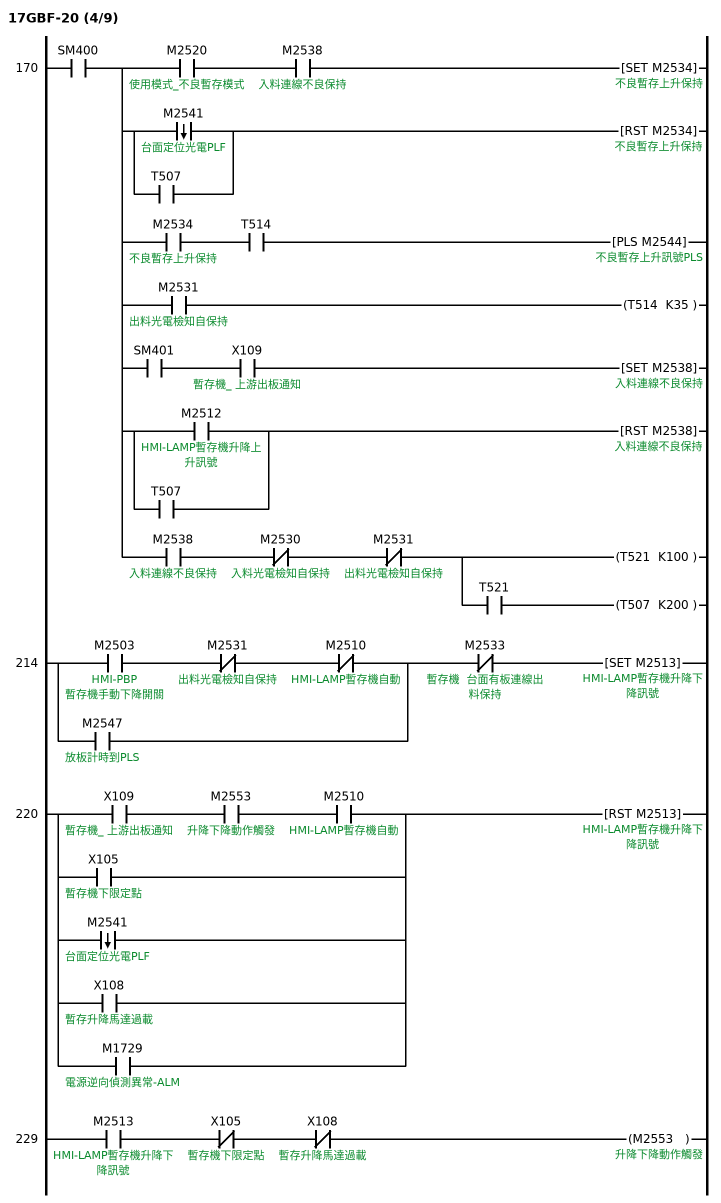
[picture p144: ladder of 17GBF-20, rungs at steps 170 to 229]
170   LD      SM400
      MPS
      AND     M2520  ; 使用模式_不良暫存模式
      AND     M2538  ; 入料連線不良保持
      SET     M2534  ; 不良暫存上升保持
      MRD
      LDF     M2541  ; 台面定位光電PLF
      OR      T507
      ANB
      RST     M2534  ; 不良暫存上升保持
      MRD
      AND     M2534  ; 不良暫存上升保持
      AND     T514
      PLS     M2544  ; 不良暫存上升訊號PLS
      MRD
      AND     M2531  ; 出料光電檢知自保持
      OUT     T514 K35
      MRD
      AND     SM401
      AND     X109  ; 暫存機_ 上游出板通知
      SET     M2538  ; 入料連線不良保持
      MRD
      LD      M2512  ; HMI-LAMP暫存機升降上升訊號
      OR      T507
      ANB
      RST     M2538  ; 入料連線不良保持
      MPP
      AND     M2538  ; 入料連線不良保持
      ANI     M2530  ; 入料光電檢知自保持
      ANI     M2531  ; 出料光電檢知自保持
      OUT     T521 K100
      AND     T521
      OUT     T507 K200
214   LD      M2503  ; HMI-PBP 暫存機手動下降開關
      ANI     M2531  ; 出料光電檢知自保持
      ANI     M2510  ; HMI-LAMP暫存機自動
      OR      M2547  ; 放板計時到PLS
      ANI     M2533  ; 暫存機  台面有板連線出料保持
      SET     M2513  ; HMI-LAMP暫存機升降下降訊號
220   LD      X109  ; 暫存機_ 上游出板通知
      AND     M2553  ; 升降下降動作觸發
      AND     M2510  ; HMI-LAMP暫存機自動
      OR      X105  ; 暫存機下限定點
      ORF     M2541  ; 台面定位光電PLF
      OR      X108  ; 暫存升降馬達過載
      OR      M1729  ; 電源逆向偵測異常-ALM
      RST     M2513  ; HMI-LAMP暫存機升降下降訊號
229   LD      M2513  ; HMI-LAMP暫存機升降下降訊號
      ANI     X105  ; 暫存機下限定點
      ANI     X108  ; 暫存升降馬達過載
      OUT     M2553  ; 升降下降動作觸發
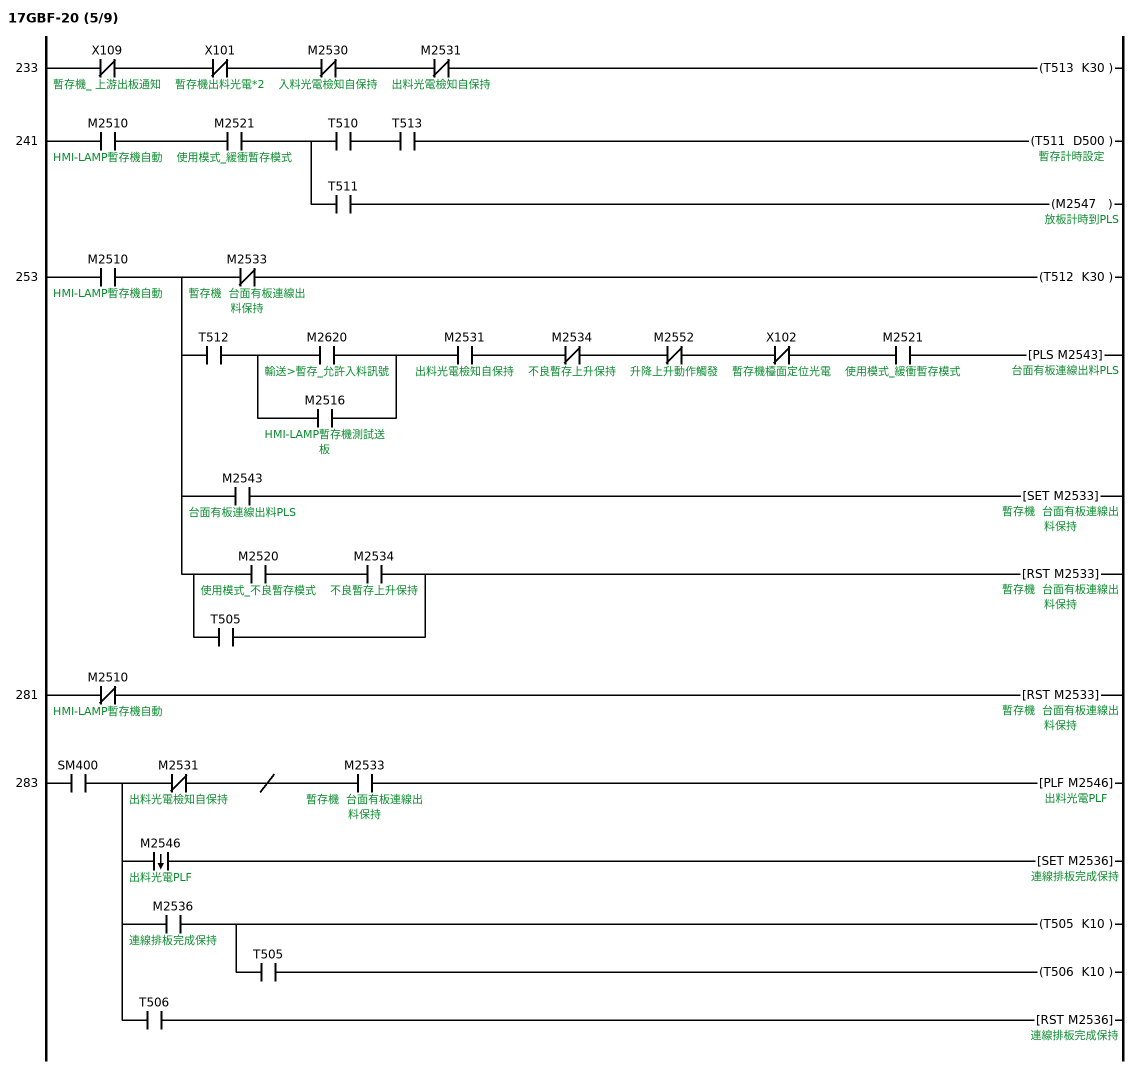
233   LDI     X109  ; 暫存機_ 上游出板通知
      ANI     X101  ; 暫存機出料光電*2
      ANI     M2530  ; 入料光電檢知自保持
      ANI     M2531  ; 出料光電檢知自保持
      OUT     T513 K30
241   LD      M2510  ; HMI-LAMP暫存機自動
      AND     M2521  ; 使用模式_緩衝暫存模式
      MPS
      AND     T510
      AND     T513
      OUT     T511 D500  ; 暫存計時設定
      MPP
      AND     T511
      OUT     M2547  ; 放板計時到PLS
253   LD      M2510  ; HMI-LAMP暫存機自動
      MPS
      ANI     M2533  ; 暫存機  台面有板連線出料保持
      OUT     T512 K30
      MRD
      AND     T512
      LD      M2620  ; 輸送>暫存_允許入料訊號
      OR      M2516  ; HMI-LAMP暫存機測試送板
      ANB
      AND     M2531  ; 出料光電檢知自保持
      ANI     M2534  ; 不良暫存上升保持
      ANI     M2552  ; 升降上升動作觸發
      ANI     X102  ; 暫存機檯面定位光電
      AND     M2521  ; 使用模式_緩衝暫存模式
      PLS     M2543  ; 台面有板連線出料PLS
      MRD
      AND     M2543  ; 台面有板連線出料PLS
      SET     M2533  ; 暫存機  台面有板連線出料保持
      MPP
      LD      M2520  ; 使用模式_不良暫存模式
      AND     M2534  ; 不良暫存上升保持
      OR      T505
      ANB
      RST     M2533  ; 暫存機  台面有板連線出料保持
281   LDI     M2510  ; HMI-LAMP暫存機自動
      RST     M2533  ; 暫存機  台面有板連線出料保持
283   LD      SM400
      MPS
      ANI     M2531  ; 出料光電檢知自保持
      INV
      AND     M2533  ; 暫存機  台面有板連線出料保持
      PLF     M2546  ; 出料光電PLF
      MRD
      ANDF    M2546  ; 出料光電PLF
      SET     M2536  ; 連線排板完成保持
      MRD
      AND     M2536  ; 連線排板完成保持
      OUT     T505 K10
      AND     T505
      OUT     T506 K10
      MPP
      AND     T506
      RST     M2536  ; 連線排板完成保持
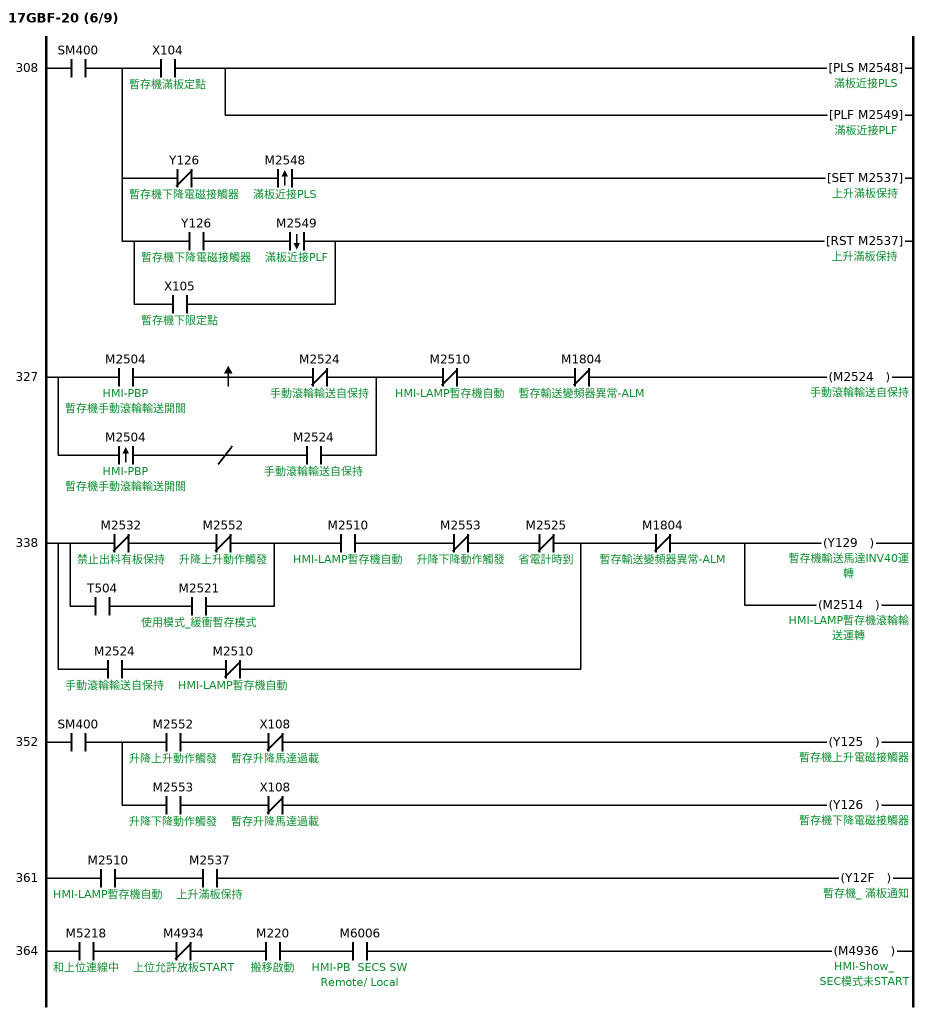
308   LD      SM400
      MPS
      AND     X104  ; 暫存機滿板定點
      PLS     M2548  ; 滿板近接PLS
      PLF     M2549  ; 滿板近接PLF
      MRD
      ANI     Y126  ; 暫存機下降電磁接觸器
      ANDP    M2548  ; 滿板近接PLS
      SET     M2537  ; 上升滿板保持
      MPP
      LD      Y126  ; 暫存機下降電磁接觸器
      ANDF    M2549  ; 滿板近接PLF
      OR      X105  ; 暫存機下限定點
      ANB
      RST     M2537  ; 上升滿板保持
327   LD      M2504  ; HMI-PBP 暫存機手動滾輪輸送開關
      MEP
      ANI     M2524  ; 手動滾輪輸送自保持
      LDP     M2504  ; HMI-PBP 暫存機手動滾輪輸送開關
      INV
      AND     M2524  ; 手動滾輪輸送自保持
      ORB
      ANI     M2510  ; HMI-LAMP暫存機自動
      ANI     M1804  ; 暫存輸送變頻器異常-ALM
      OUT     M2524  ; 手動滾輪輸送自保持
338   LDI     M2532  ; 禁止出料有板保持
      ANI     M2552  ; 升降上升動作觸發
      LD      T504
      AND     M2521  ; 使用模式_緩衝暫存模式
      ORB
      AND     M2510  ; HMI-LAMP暫存機自動
      ANI     M2553  ; 升降下降動作觸發
      ANI     M2525  ; 省電計時到
      LD      M2524  ; 手動滾輪輸送自保持
      ANI     M2510  ; HMI-LAMP暫存機自動
      ORB
      ANI     M1804  ; 暫存輸送變頻器異常-ALM
      OUT     Y129  ; 暫存機輸送馬達INV40運轉
      OUT     M2514  ; HMI-LAMP暫存機滾輪輸送運轉
352   LD      SM400
      MPS
      AND     M2552  ; 升降上升動作觸發
      ANI     X108  ; 暫存升降馬達過載
      OUT     Y125  ; 暫存機上升電磁接觸器
      MPP
      AND     M2553  ; 升降下降動作觸發
      ANI     X108  ; 暫存升降馬達過載
      OUT     Y126  ; 暫存機下降電磁接觸器
361   LD      M2510  ; HMI-LAMP暫存機自動
      AND     M2537  ; 上升滿板保持
      OUT     Y12F  ; 暫存機_ 滿板通知
364   LD      M5218  ; 和上位連線中
      ANI     M4934  ; 上位允許放板START
      AND     M220  ; 搬移啟動
      AND     M6006  ; HMI-PB  SECS SW  Remote/ Local
      OUT     M4936  ; HMI-Show_SEC模式未START
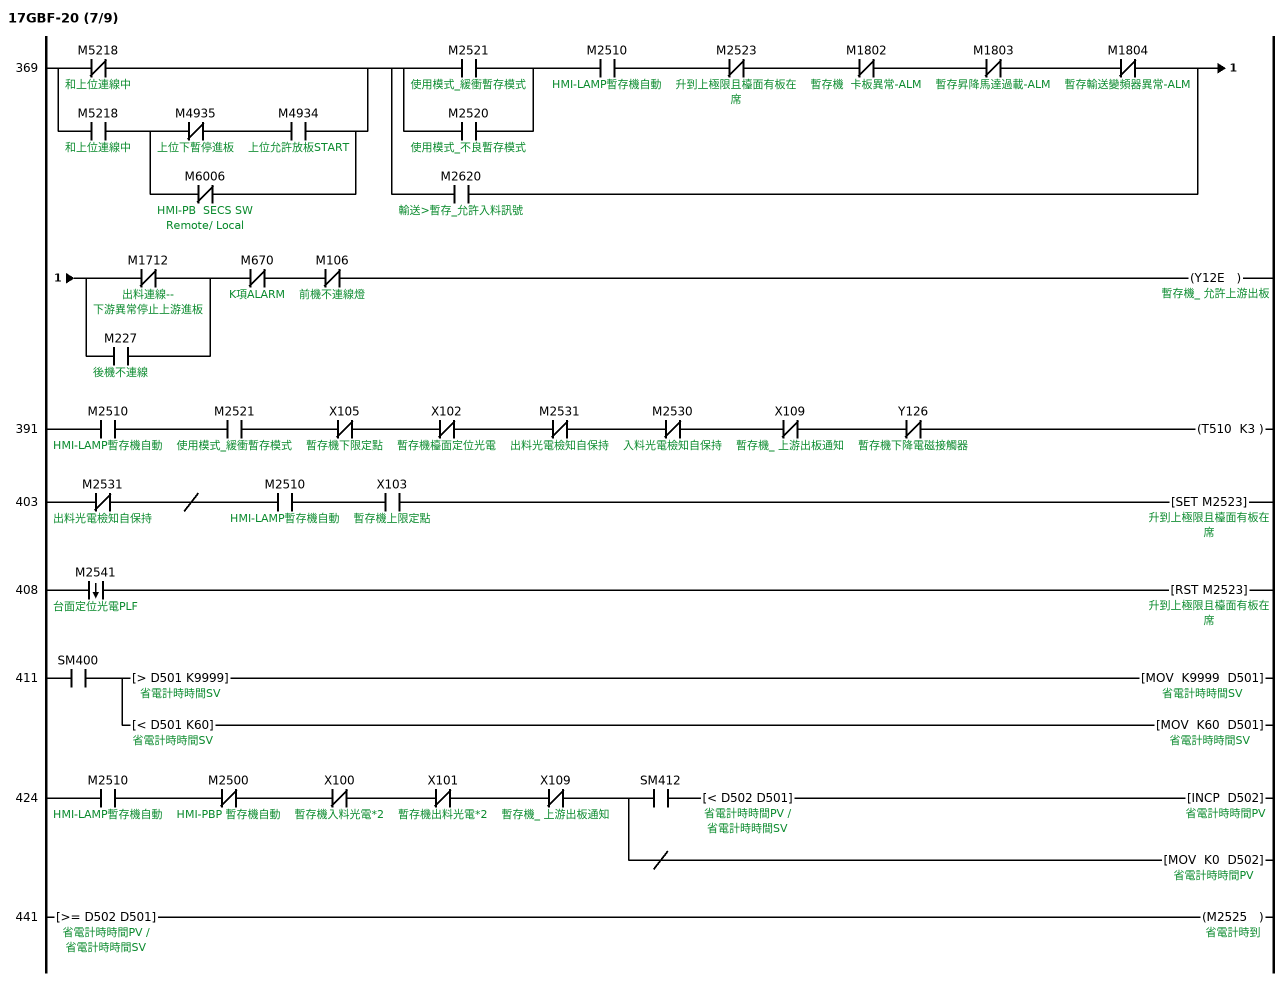
369   LDI     M5218  ; 和上位連線中
      LD      M5218  ; 和上位連線中
      LDI     M4935  ; 上位下暫停進板
      AND     M4934  ; 上位允許放板START
      ORI     M6006  ; HMI-PB  SECS SW  Remote/ Local
      ANB
      ORB
      LD      M2521  ; 使用模式_緩衝暫存模式
      OR      M2520  ; 使用模式_不良暫存模式
      AND     M2510  ; HMI-LAMP暫存機自動
      ANI     M2523  ; 升到上極限且檯面有板在席
      ANI     M1802  ; 暫存機  卡板異常-ALM
      ANI     M1803  ; 暫存昇降馬達過載-ALM
      ANI     M1804  ; 暫存輸送變頻器異常-ALM
      OR      M2620  ; 輸送>暫存_允許入料訊號
      ANB
      LDI     M1712  ; 出料連線--下游異常停止上游進板
      OR      M227  ; 後機不連線
      ANB
      ANI     M670  ; K項ALARM
      ANI     M106  ; 前機不連線燈
      OUT     Y12E  ; 暫存機_ 允許上游出板
391   LD      M2510  ; HMI-LAMP暫存機自動
      AND     M2521  ; 使用模式_緩衝暫存模式
      ANI     X105  ; 暫存機下限定點
      ANI     X102  ; 暫存機檯面定位光電
      ANI     M2531  ; 出料光電檢知自保持
      ANI     M2530  ; 入料光電檢知自保持
      ANI     X109  ; 暫存機_ 上游出板通知
      ANI     Y126  ; 暫存機下降電磁接觸器
      OUT     T510 K3
403   LDI     M2531  ; 出料光電檢知自保持
      INV
      AND     M2510  ; HMI-LAMP暫存機自動
      AND     X103  ; 暫存機上限定點
      SET     M2523  ; 升到上極限且檯面有板在席
408   LDF     M2541  ; 台面定位光電PLF
      RST     M2523  ; 升到上極限且檯面有板在席
411   LD      SM400
      MPS
      AND>    D501 K9999  ; 省電計時時間SV
      MOV     K9999 D501
      MPP
      AND<    D501 K60  ; 省電計時時間SV
      MOV     K60 D501
424   LD      M2510  ; HMI-LAMP暫存機自動
      ANI     M2500  ; HMI-PBP 暫存機自動
      ANI     X100  ; 暫存機入料光電*2
      ANI     X101  ; 暫存機出料光電*2
      ANI     X109  ; 暫存機_ 上游出板通知
      MPS
      AND     SM412
      AND<    D502 D501  ; 省電計時時間PV / 省電計時時間SV
      INCP    D502
      MPP
      INV
      MOV     K0 D502
441   LD>=    D502 D501  ; 省電計時時間PV / 省電計時時間SV
      OUT     M2525  ; 省電計時到
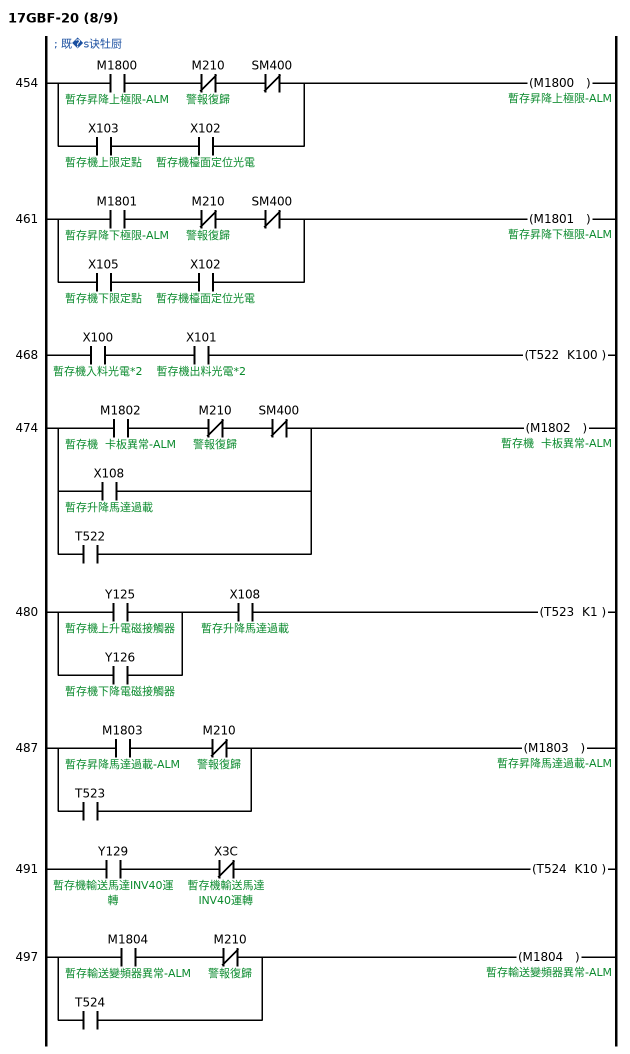
; 暫存機警報
454   LD      M1800  ; 暫存昇降上極限-ALM
      ANI     M210  ; 警報復歸
      ANI     SM400
      LD      X103  ; 暫存機上限定點
      AND     X102  ; 暫存機檯面定位光電
      ORB
      OUT     M1800  ; 暫存昇降上極限-ALM
461   LD      M1801  ; 暫存昇降下極限-ALM
      ANI     M210  ; 警報復歸
      ANI     SM400
      LD      X105  ; 暫存機下限定點
      AND     X102  ; 暫存機檯面定位光電
      ORB
      OUT     M1801  ; 暫存昇降下極限-ALM
468   LD      X100  ; 暫存機入料光電*2
      AND     X101  ; 暫存機出料光電*2
      OUT     T522 K100
474   LD      M1802  ; 暫存機  卡板異常-ALM
      ANI     M210  ; 警報復歸
      ANI     SM400
      OR      X108  ; 暫存升降馬達過載
      OR      T522
      OUT     M1802  ; 暫存機  卡板異常-ALM
480   LD      Y125  ; 暫存機上升電磁接觸器
      OR      Y126  ; 暫存機下降電磁接觸器
      AND     X108  ; 暫存升降馬達過載
      OUT     T523 K1
487   LD      M1803  ; 暫存昇降馬達過載-ALM
      ANI     M210  ; 警報復歸
      OR      T523
      OUT     M1803  ; 暫存昇降馬達過載-ALM
491   LD      Y129  ; 暫存機輸送馬達INV40運轉
      ANI     X3C  ; 暫存機輸送馬達  INV40運轉
      OUT     T524 K10
497   LD      M1804  ; 暫存輸送變頻器異常-ALM
      ANI     M210  ; 警報復歸
      OR      T524
      OUT     M1804  ; 暫存輸送變頻器異常-ALM
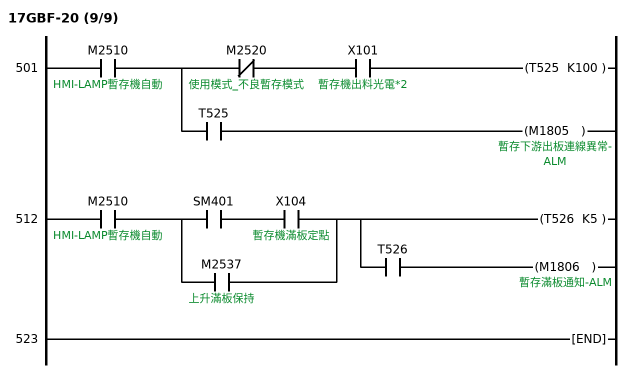
501   LD      M2510  ; HMI-LAMP暫存機自動
      MPS
      ANI     M2520  ; 使用模式_不良暫存模式
      AND     X101  ; 暫存機出料光電*2
      OUT     T525 K100
      MPP
      AND     T525
      OUT     M1805  ; 暫存下游出板連線異常-ALM
512   LD      M2510  ; HMI-LAMP暫存機自動
      LD      SM401
      AND     X104  ; 暫存機滿板定點
      OR      M2537  ; 上升滿板保持
      ANB
      OUT     T526 K5
      AND     T526
      OUT     M1806  ; 暫存滿板通知-ALM
523   END
END_PROGRAM

PROGRAM 18GCV
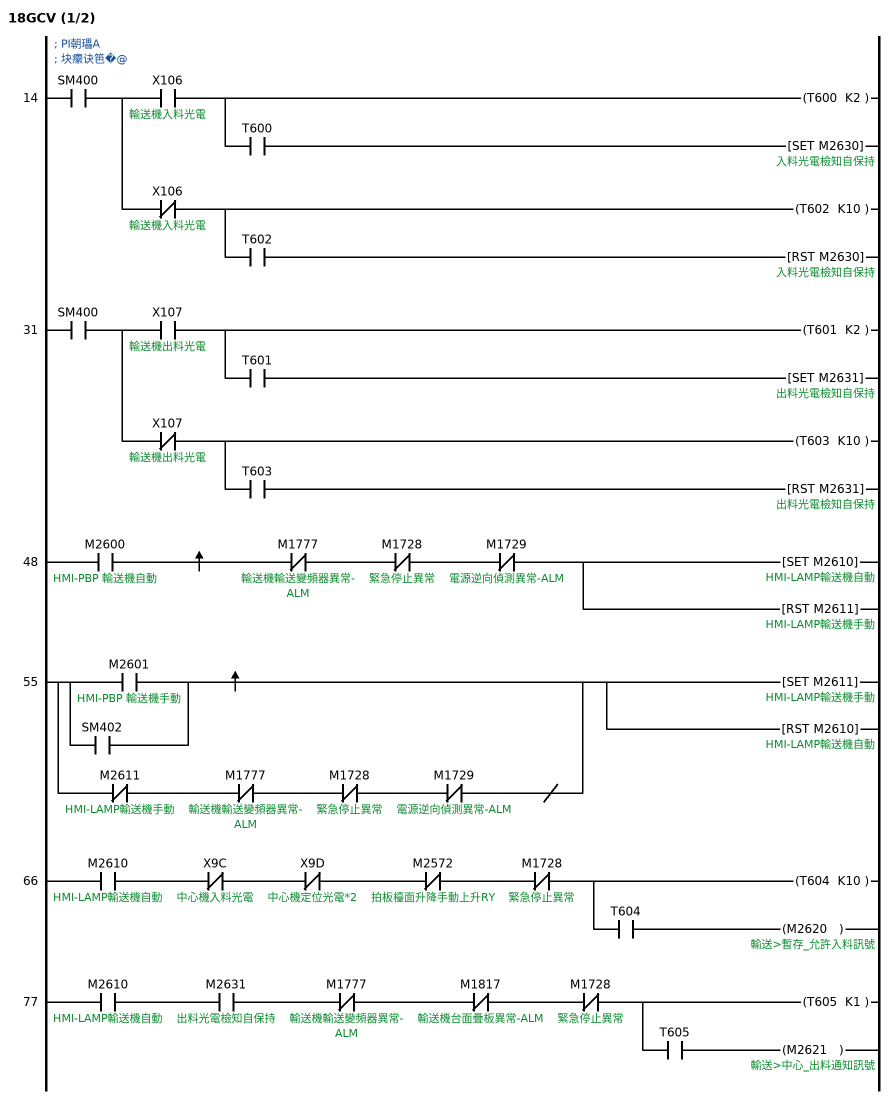
; PI朝瓃Α
; 輸送機動作
14    LD      SM400
      MPS
      AND     X106  ; 輸送機入料光電
      OUT     T600 K2
      AND     T600
      SET     M2630  ; 入料光電檢知自保持
      MPP
      ANI     X106  ; 輸送機入料光電
      OUT     T602 K10
      AND     T602
      RST     M2630  ; 入料光電檢知自保持
31    LD      SM400
      MPS
      AND     X107  ; 輸送機出料光電
      OUT     T601 K2
      AND     T601
      SET     M2631  ; 出料光電檢知自保持
      MPP
      ANI     X107  ; 輸送機出料光電
      OUT     T603 K10
      AND     T603
      RST     M2631  ; 出料光電檢知自保持
48    LD      M2600  ; HMI-PBP 輸送機自動
      MEP
      ANI     M1777  ; 輸送機輸送變頻器異常-ALM
      ANI     M1728  ; 緊急停止異常
      ANI     M1729  ; 電源逆向偵測異常-ALM
      SET     M2610  ; HMI-LAMP輸送機自動
      RST     M2611  ; HMI-LAMP輸送機手動
55    LD      M2601  ; HMI-PBP 輸送機手動
      OR      SM402
      MEP
      LDI     M2611  ; HMI-LAMP輸送機手動
      ANI     M1777  ; 輸送機輸送變頻器異常-ALM
      ANI     M1728  ; 緊急停止異常
      ANI     M1729  ; 電源逆向偵測異常-ALM
      INV
      ORB
      SET     M2611  ; HMI-LAMP輸送機手動
      RST     M2610  ; HMI-LAMP輸送機自動
66    LD      M2610  ; HMI-LAMP輸送機自動
      ANI     X9C  ; 中心機入料光電
      ANI     X9D  ; 中心機定位光電*2
      ANI     M2572  ; 拍板檯面升降手動上升RY
      ANI     M1728  ; 緊急停止異常
      OUT     T604 K10
      AND     T604
      OUT     M2620  ; 輸送>暫存_允許入料訊號
77    LD      M2610  ; HMI-LAMP輸送機自動
      AND     M2631  ; 出料光電檢知自保持
      ANI     M1777  ; 輸送機輸送變頻器異常-ALM
      ANI     M1817  ; 輸送機台面疊板異常-ALM
      ANI     M1728  ; 緊急停止異常
      OUT     T605 K1
      AND     T605
      OUT     M2621  ; 輸送>中心_出料通知訊號
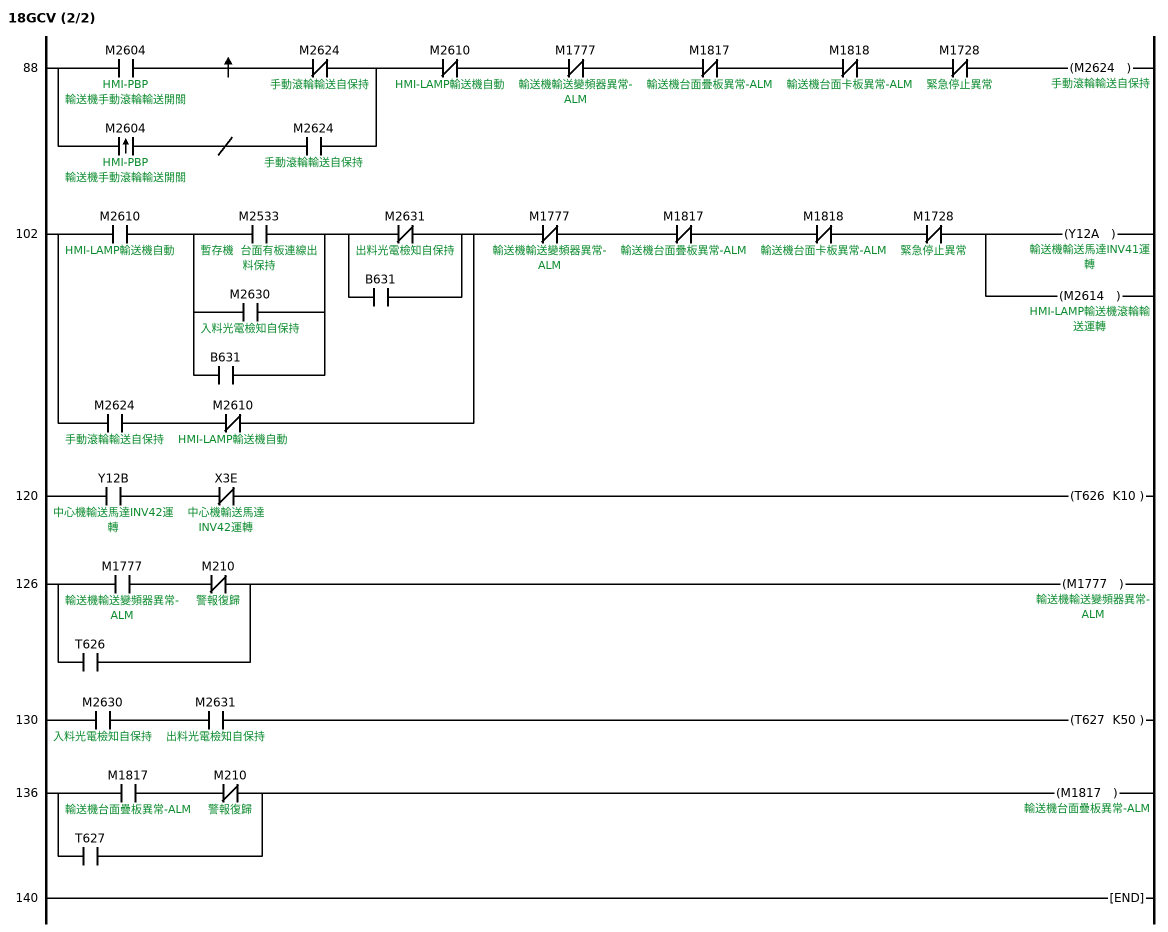
88    LD      M2604  ; HMI-PBP 輸送機手動滾輪輸送開關
      MEP
      ANI     M2624  ; 手動滾輪輸送自保持
      LDP     M2604  ; HMI-PBP 輸送機手動滾輪輸送開關
      INV
      AND     M2624  ; 手動滾輪輸送自保持
      ORB
      ANI     M2610  ; HMI-LAMP輸送機自動
      ANI     M1777  ; 輸送機輸送變頻器異常-ALM
      ANI     M1817  ; 輸送機台面疊板異常-ALM
      ANI     M1818  ; 輸送機台面卡板異常-ALM
      ANI     M1728  ; 緊急停止異常
      OUT     M2624  ; 手動滾輪輸送自保持
102   LD      M2610  ; HMI-LAMP輸送機自動
      LD      M2533  ; 暫存機  台面有板連線出料保持
      OR      M2630  ; 入料光電檢知自保持
      OR      B631
      ANB
      LDI     M2631  ; 出料光電檢知自保持
      OR      B631
      ANB
      LD      M2624  ; 手動滾輪輸送自保持
      ANI     M2610  ; HMI-LAMP輸送機自動
      ORB
      ANI     M1777  ; 輸送機輸送變頻器異常-ALM
      ANI     M1817  ; 輸送機台面疊板異常-ALM
      ANI     M1818  ; 輸送機台面卡板異常-ALM
      ANI     M1728  ; 緊急停止異常
      OUT     Y12A  ; 輸送機輸送馬達INV41運轉
      OUT     M2614  ; HMI-LAMP輸送機滾輪輸送運轉
120   LD      Y12B  ; 中心機輸送馬達INV42運轉
      ANI     X3E  ; 中心機輸送馬達  INV42運轉
      OUT     T626 K10
126   LD      M1777  ; 輸送機輸送變頻器異常-ALM
      ANI     M210  ; 警報復歸
      OR      T626
      OUT     M1777  ; 輸送機輸送變頻器異常-ALM
130   LD      M2630  ; 入料光電檢知自保持
      AND     M2631  ; 出料光電檢知自保持
      OUT     T627 K50
136   LD      M1817  ; 輸送機台面疊板異常-ALM
      ANI     M210  ; 警報復歸
      OR      T627
      OUT     M1817  ; 輸送機台面疊板異常-ALM
140   END
END_PROGRAM

PROGRAM 19GTC-7
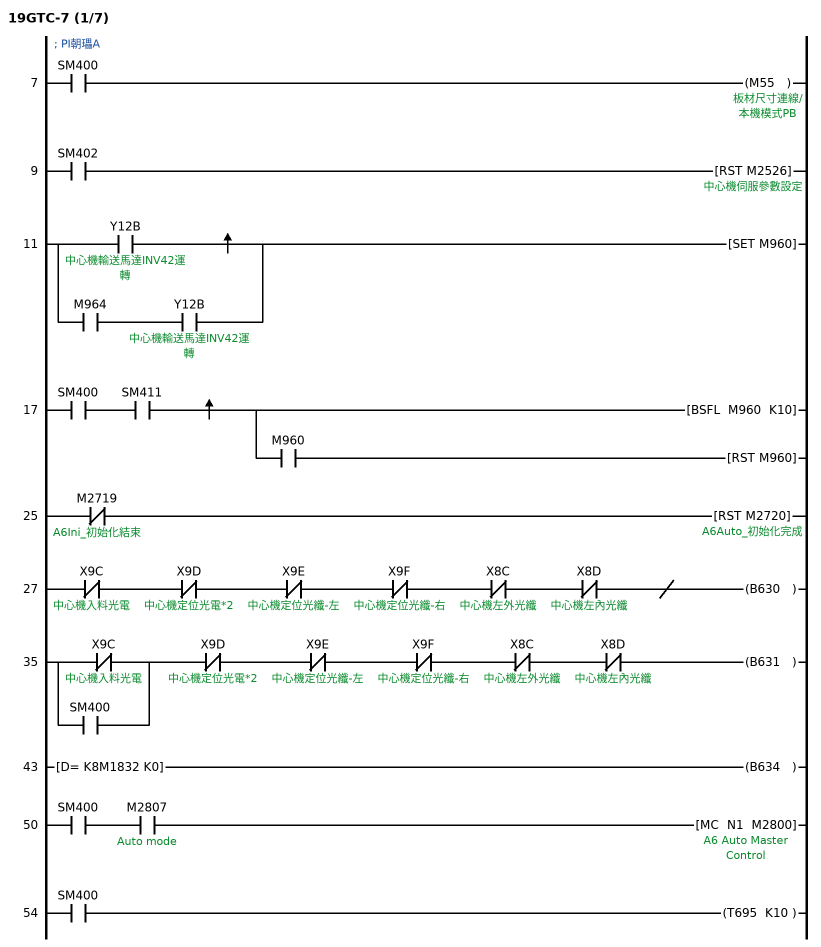
; PI朝瓃Α
7     LD      SM400
      OUT     M55  ; 板材尺寸連線/本機模式PB
9     LD      SM402
      RST     M2526  ; 中心機伺服參數設定
11    LD      Y12B  ; 中心機輸送馬達INV42運轉
      MEP
      LD      M964
      AND     Y12B  ; 中心機輸送馬達INV42運轉
      ORB
      SET     M960
17    LD      SM400
      AND     SM411
      MEP
      BSFL    M960 K10
      AND     M960
      RST     M960
25    LDI     M2719  ; A6Ini_初始化結束
      RST     M2720  ; A6Auto_初始化完成
27    LDI     X9C  ; 中心機入料光電
      ANI     X9D  ; 中心機定位光電*2
      ANI     X9E  ; 中心機定位光纖-左
      ANI     X9F  ; 中心機定位光纖-右
      ANI     X8C  ; 中心機左外光纖
      ANI     X8D  ; 中心機左內光纖
      INV
      OUT     B630
35    LDI     X9C  ; 中心機入料光電
      OR      SM400
      ANI     X9D  ; 中心機定位光電*2
      ANI     X9E  ; 中心機定位光纖-左
      ANI     X9F  ; 中心機定位光纖-右
      ANI     X8C  ; 中心機左外光纖
      ANI     X8D  ; 中心機左內光纖
      OUT     B631
43    LDD=    K8M1832 K0
      OUT     B634
50    LD      SM400
      AND     M2807  ; Auto mode
      MC      N1 M2800  ; A6 Auto Master Control
54    LD      SM400
      OUT     T695 K10
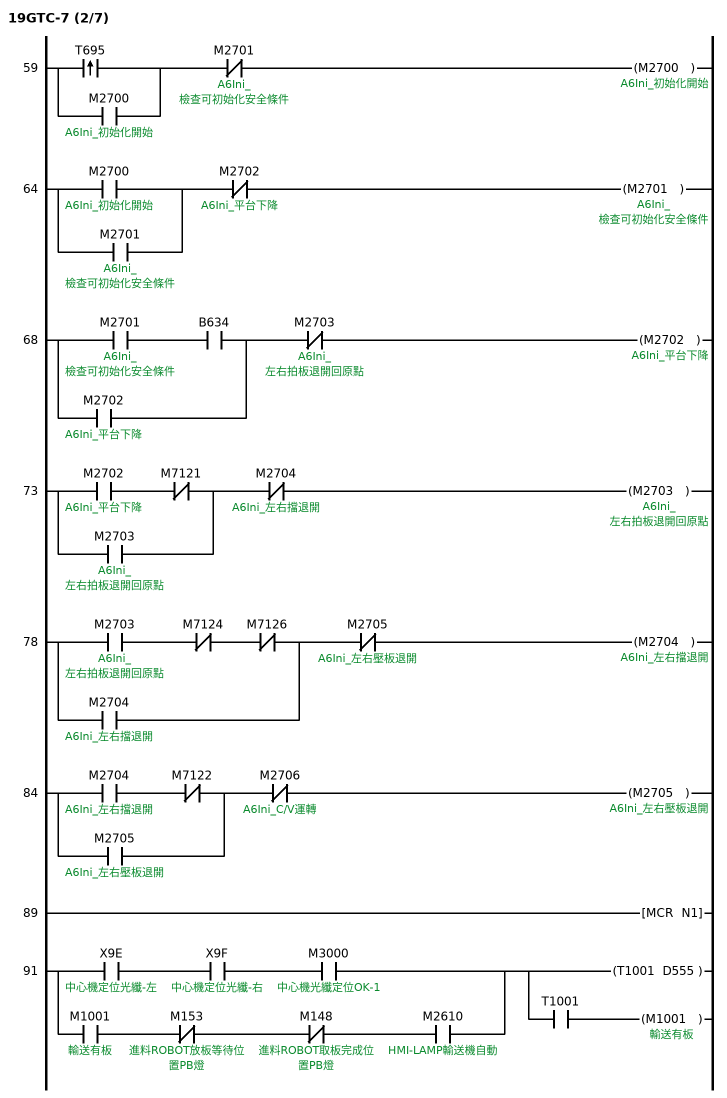
59    LDP     T695
      OR      M2700  ; A6Ini_初始化開始
      ANI     M2701  ; A6Ini_檢查可初始化安全條件
      OUT     M2700  ; A6Ini_初始化開始
64    LD      M2700  ; A6Ini_初始化開始
      OR      M2701  ; A6Ini_檢查可初始化安全條件
      ANI     M2702  ; A6Ini_平台下降
      OUT     M2701  ; A6Ini_檢查可初始化安全條件
68    LD      M2701  ; A6Ini_檢查可初始化安全條件
      AND     B634
      OR      M2702  ; A6Ini_平台下降
      ANI     M2703  ; A6Ini_左右拍板退開回原點
      OUT     M2702  ; A6Ini_平台下降
73    LD      M2702  ; A6Ini_平台下降
      ANI     M7121
      OR      M2703  ; A6Ini_左右拍板退開回原點
      ANI     M2704  ; A6Ini_左右擋退開
      OUT     M2703  ; A6Ini_左右拍板退開回原點
78    LD      M2703  ; A6Ini_左右拍板退開回原點
      ANI     M7124
      ANI     M7126
      OR      M2704  ; A6Ini_左右擋退開
      ANI     M2705  ; A6Ini_左右壓板退開
      OUT     M2704  ; A6Ini_左右擋退開
84    LD      M2704  ; A6Ini_左右擋退開
      ANI     M7122
      OR      M2705  ; A6Ini_左右壓板退開
      ANI     M2706  ; A6Ini_C/V運轉
      OUT     M2705  ; A6Ini_左右壓板退開
89    MCR     N1
91    LD      X9E  ; 中心機定位光纖-左
      AND     X9F  ; 中心機定位光纖-右
      AND     M3000  ; 中心機光纖定位OK-1
      LD      M1001  ; 輸送有板
      ANI     M153  ; 進料ROBOT放板等待位置PB燈
      ANI     M148  ; 進料ROBOT取板完成位置PB燈
      AND     M2610  ; HMI-LAMP輸送機自動
      ORB
      OUT     T1001 D555
      AND     T1001
      OUT     M1001  ; 輸送有板
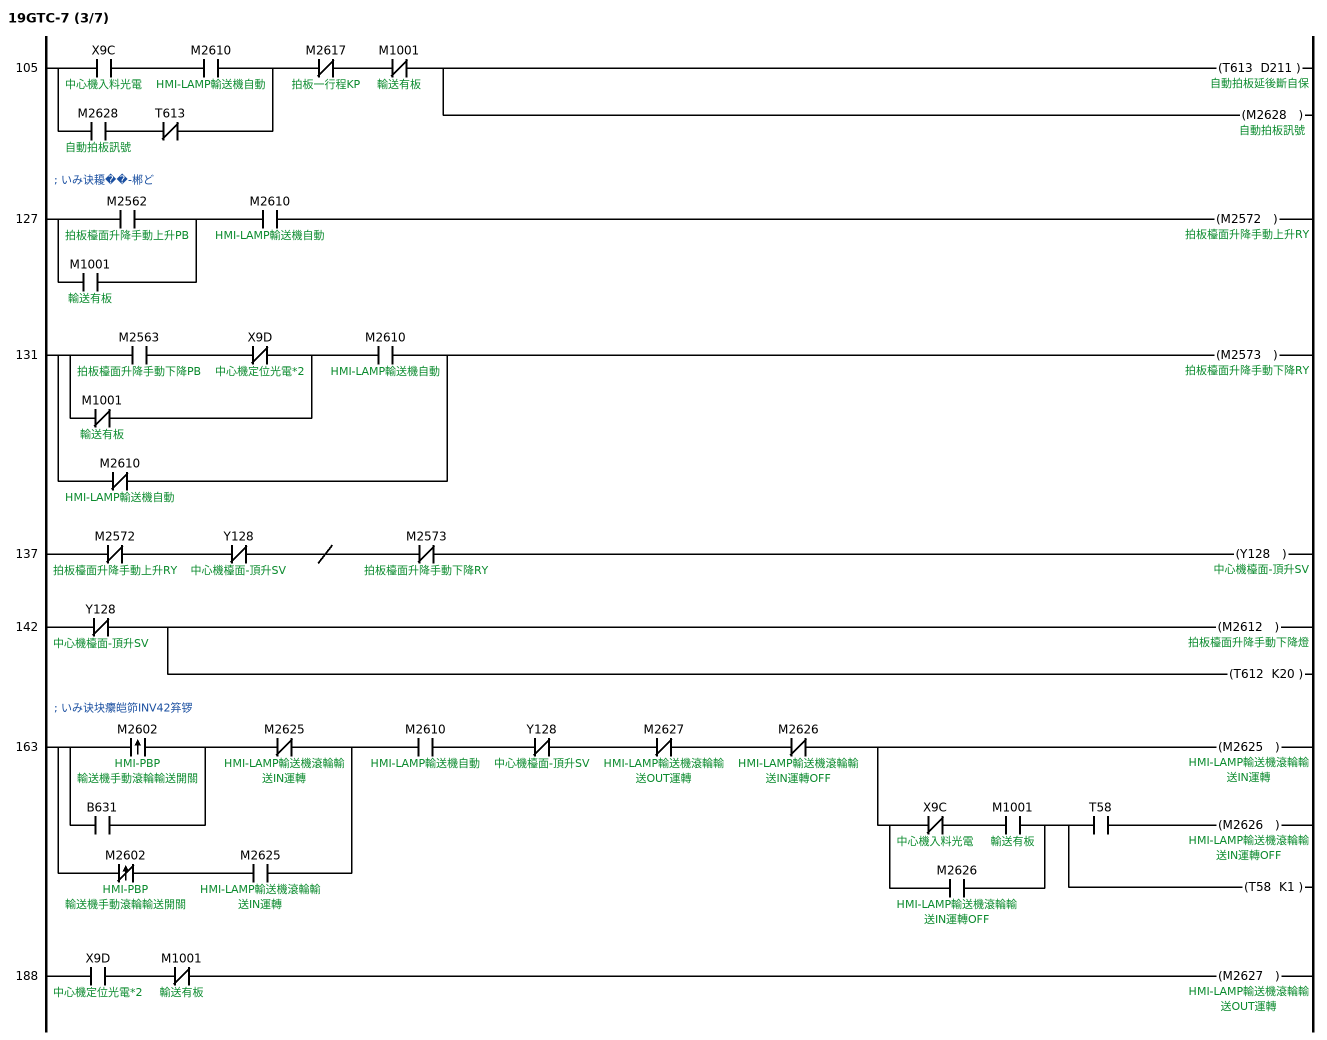
105   LD      X9C  ; 中心機入料光電
      AND     M2610  ; HMI-LAMP輸送機自動
      LD      M2628  ; 自動拍板訊號
      ANI     T613
      ORB
      ANI     M2617  ; 拍板一行程KP
      ANI     M1001  ; 輸送有板
      OUT     T613 D211  ; 自動拍板延後斷自保
      OUT     M2628  ; 自動拍板訊號
; 中心機檯面-頂升
127   LD      M2562  ; 拍板檯面升降手動上升PB
      OR      M1001  ; 輸送有板
      AND     M2610  ; HMI-LAMP輸送機自動
      OUT     M2572  ; 拍板檯面升降手動上升RY
131   LD      M2563  ; 拍板檯面升降手動下降PB
      ANI     X9D  ; 中心機定位光電*2
      ORI     M1001  ; 輸送有板
      AND     M2610  ; HMI-LAMP輸送機自動
      ORI     M2610  ; HMI-LAMP輸送機自動
      OUT     M2573  ; 拍板檯面升降手動下降RY
137   LDI     M2572  ; 拍板檯面升降手動上升RY
      ANI     Y128  ; 中心機檯面-頂升SV
      INV
      ANI     M2573  ; 拍板檯面升降手動下降RY
      OUT     Y128  ; 中心機檯面-頂升SV
142   LDI     Y128  ; 中心機檯面-頂升SV
      OUT     M2612  ; 拍板檯面升降手動下降燈
      OUT     T612 K20
; 中心機輸送馬達INV42運轉
163   LDP     M2602  ; HMI-PBP 輸送機手動滾輪輸送開關
      OR      B631
      ANI     M2625  ; HMI-LAMP輸送機滾輪輸送IN運轉
      LDPI    M2602  ; HMI-PBP 輸送機手動滾輪輸送開關
      AND     M2625  ; HMI-LAMP輸送機滾輪輸送IN運轉
      ORB
      AND     M2610  ; HMI-LAMP輸送機自動
      ANI     Y128  ; 中心機檯面-頂升SV
      ANI     M2627  ; HMI-LAMP輸送機滾輪輸送OUT運轉
      ANI     M2626  ; HMI-LAMP輸送機滾輪輸送IN運轉OFF
      OUT     M2625  ; HMI-LAMP輸送機滾輪輸送IN運轉
      LDI     X9C  ; 中心機入料光電
      AND     M1001  ; 輸送有板
      OR      M2626  ; HMI-LAMP輸送機滾輪輸送IN運轉OFF
      ANB
      MPS
      AND     T58
      OUT     M2626  ; HMI-LAMP輸送機滾輪輸送IN運轉OFF
      MPP
      OUT     T58 K1
188   LD      X9D  ; 中心機定位光電*2
      ANI     M1001  ; 輸送有板
      OUT     M2627  ; HMI-LAMP輸送機滾輪輸送OUT運轉
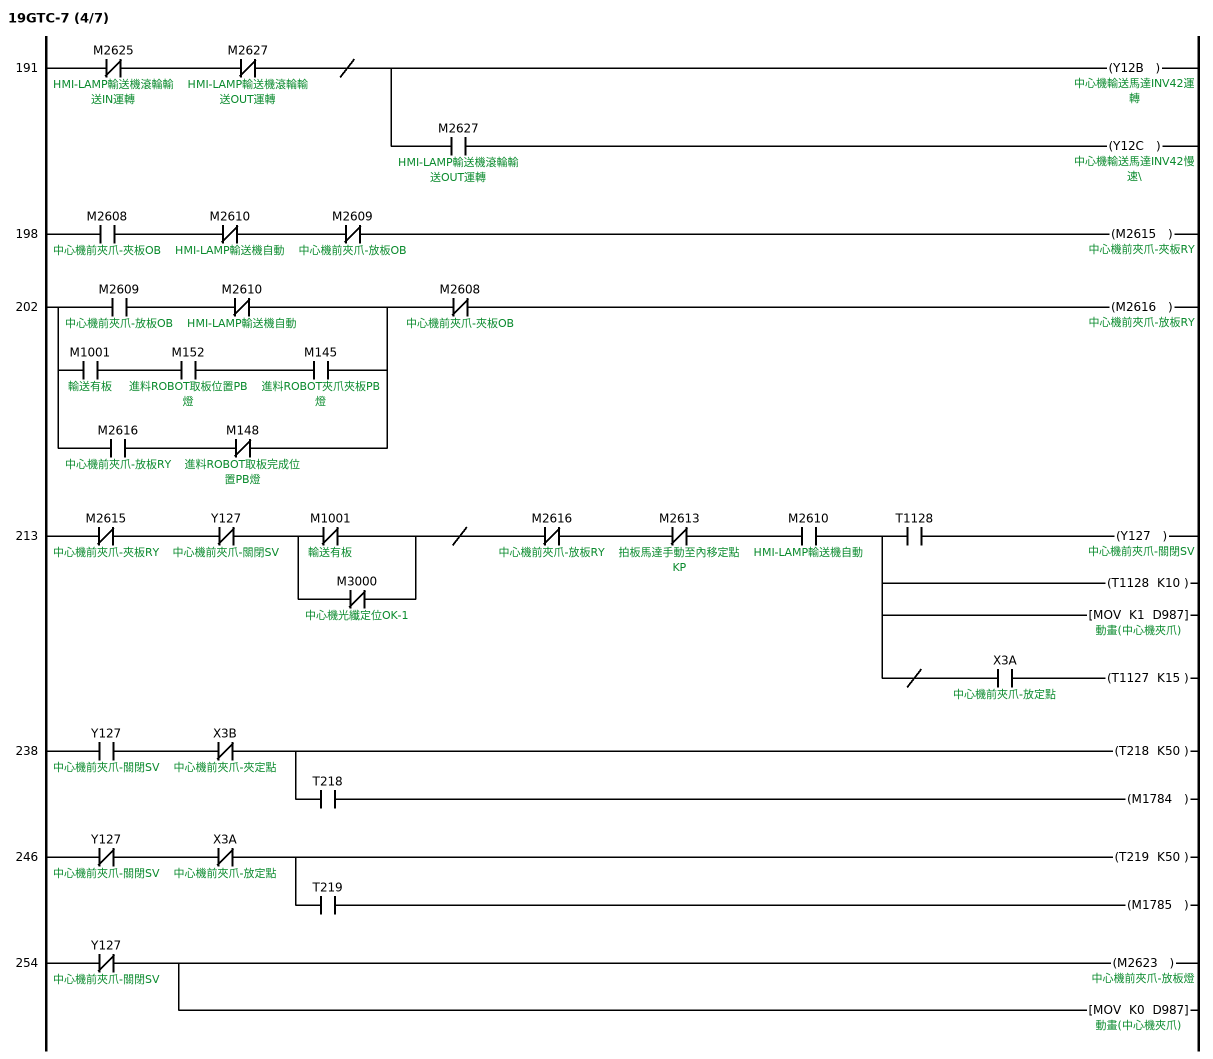
191   LDI     M2625  ; HMI-LAMP輸送機滾輪輸送IN運轉
      ANI     M2627  ; HMI-LAMP輸送機滾輪輸送OUT運轉
      INV
      OUT     Y12B  ; 中心機輸送馬達INV42運轉
      AND     M2627  ; HMI-LAMP輸送機滾輪輸送OUT運轉
      OUT     Y12C  ; 中心機輸送馬達INV42慢速\
198   LD      M2608  ; 中心機前夾爪-夾板OB
      ANI     M2610  ; HMI-LAMP輸送機自動
      ANI     M2609  ; 中心機前夾爪-放板OB
      OUT     M2615  ; 中心機前夾爪-夾板RY
202   LD      M2609  ; 中心機前夾爪-放板OB
      ANI     M2610  ; HMI-LAMP輸送機自動
      LD      M1001  ; 輸送有板
      AND     M152  ; 進料ROBOT取板位置PB燈
      AND     M145  ; 進料ROBOT夾爪夾板PB燈
      ORB
      LD      M2616  ; 中心機前夾爪-放板RY
      ANI     M148  ; 進料ROBOT取板完成位置PB燈
      ORB
      ANI     M2608  ; 中心機前夾爪-夾板OB
      OUT     M2616  ; 中心機前夾爪-放板RY
213   LDI     M2615  ; 中心機前夾爪-夾板RY
      ANI     Y127  ; 中心機前夾爪-關閉SV
      LDI     M1001  ; 輸送有板
      ORI     M3000  ; 中心機光纖定位OK-1
      ANB
      INV
      ANI     M2616  ; 中心機前夾爪-放板RY
      ANI     M2613  ; 拍板馬達手動至內移定點KP
      AND     M2610  ; HMI-LAMP輸送機自動
      MPS
      AND     T1128
      OUT     Y127  ; 中心機前夾爪-關閉SV
      MPP
      OUT     T1128 K10
      MOV     K1 D987  ; 動畫(中心機夾爪)
      INV
      AND     X3A  ; 中心機前夾爪-放定點
      OUT     T1127 K15
238   LD      Y127  ; 中心機前夾爪-關閉SV
      ANI     X3B  ; 中心機前夾爪-夾定點
      OUT     T218 K50
      AND     T218
      OUT     M1784
246   LDI     Y127  ; 中心機前夾爪-關閉SV
      ANI     X3A  ; 中心機前夾爪-放定點
      OUT     T219 K50
      AND     T219
      OUT     M1785
254   LDI     Y127  ; 中心機前夾爪-關閉SV
      OUT     M2623  ; 中心機前夾爪-放板燈
      MOV     K0 D987
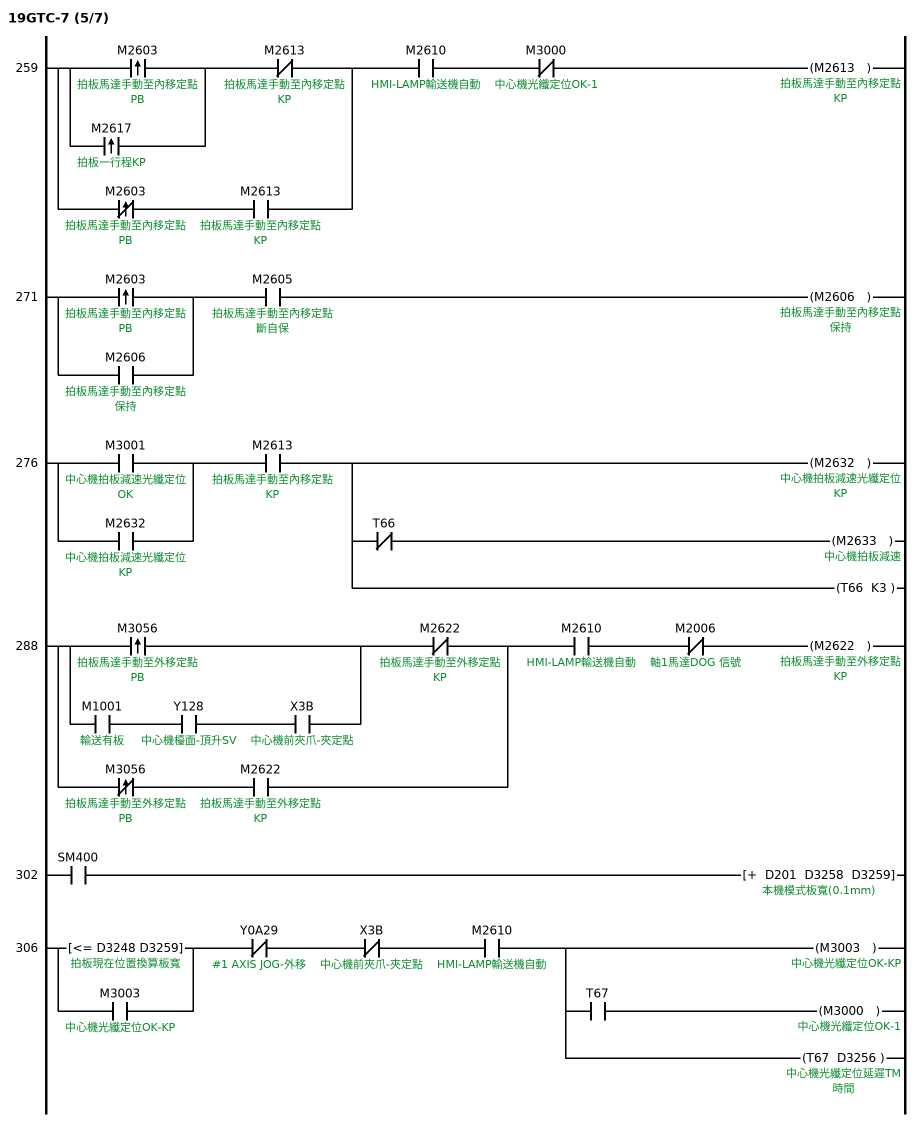
259   LDP     M2603  ; 拍板馬達手動至內移定點PB
      ORP     M2617  ; 拍板一行程KP
      ANI     M2613  ; 拍板馬達手動至內移定點KP
      LDPI    M2603  ; 拍板馬達手動至內移定點PB
      AND     M2613  ; 拍板馬達手動至內移定點KP
      ORB
      AND     M2610  ; HMI-LAMP輸送機自動
      ANI     M3000  ; 中心機光纖定位OK-1
      OUT     M2613  ; 拍板馬達手動至內移定點KP
271   LDP     M2603  ; 拍板馬達手動至內移定點PB
      OR      M2606  ; 拍板馬達手動至內移定點保持
      AND     M2605  ; 拍板馬達手動至內移定點斷自保
      OUT     M2606  ; 拍板馬達手動至內移定點保持
276   LD      M3001  ; 中心機拍板減速光纖定位OK
      OR      M2632  ; 中心機拍板減速光纖定位KP
      AND     M2613  ; 拍板馬達手動至內移定點KP
      OUT     M2632  ; 中心機拍板減速光纖定位KP
      MPS
      ANI     T66
      OUT     M2633  ; 中心機拍板減速
      MPP
      OUT     T66 K3
288   LDP     M3056  ; 拍板馬達手動至外移定點PB
      LD      M1001  ; 輸送有板
      AND     Y128  ; 中心機檯面-頂升SV
      AND     X3B  ; 中心機前夾爪-夾定點
      ORB
      ANI     M2622  ; 拍板馬達手動至外移定點KP
      LDPI    M3056  ; 拍板馬達手動至外移定點PB
      AND     M2622  ; 拍板馬達手動至外移定點KP
      ORB
      AND     M2610  ; HMI-LAMP輸送機自動
      ANI     M2006  ; 軸1馬達DOG 信號
      OUT     M2622  ; 拍板馬達手動至外移定點KP
302   LD      SM400
      +       D201 D3258 D3259  ; 本機模式板寬(0.1mm)
306   LD<=    D3248 D3259  ; 拍板現在位置換算板寬
      OR      M3003  ; 中心機光纖定位OK-KP
      ANI     Y0A29  ; #1 AXIS JOG-外移
      ANI     X3B  ; 中心機前夾爪-夾定點
      AND     M2610  ; HMI-LAMP輸送機自動
      OUT     M3003  ; 中心機光纖定位OK-KP
      MPS
      AND     T67
      OUT     M3000  ; 中心機光纖定位OK-1
      MPP
      OUT     T67 D3256  ; 中心機光纖定位延遲TM時間
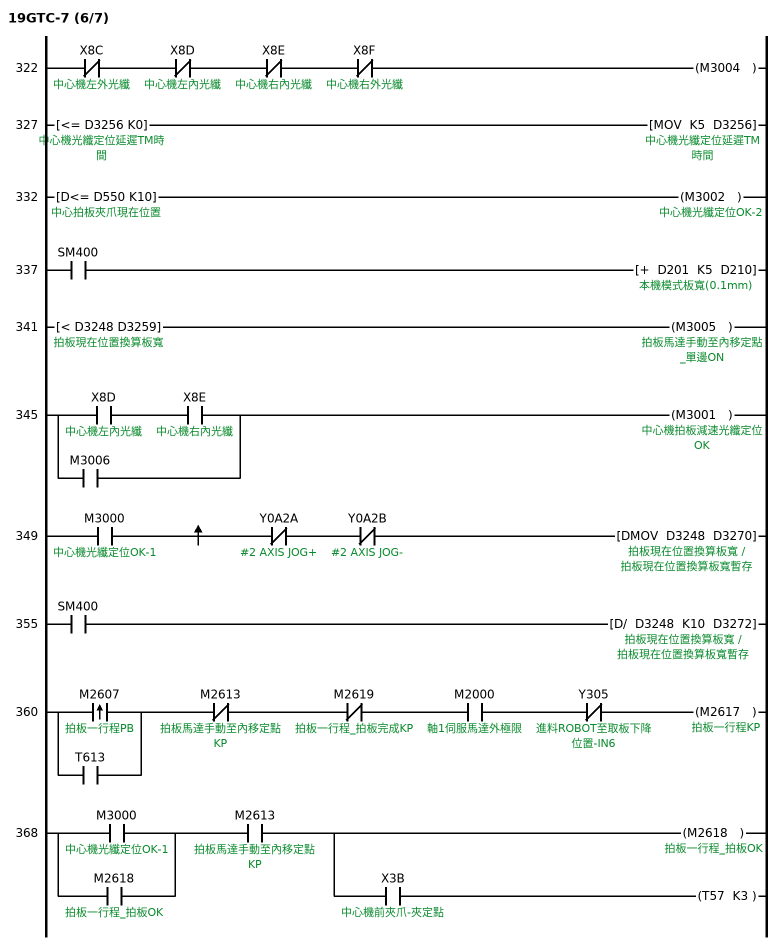
322   LDI     X8C  ; 中心機左外光纖
      ANI     X8D  ; 中心機左內光纖
      ANI     X8E  ; 中心機右內光纖
      ANI     X8F  ; 中心機右外光纖
      OUT     M3004
327   LD<=    D3256 K0  ; 中心機光纖定位延遲TM時間
      MOV     K5 D3256
332   LDD<=   D550 K10  ; 中心拍板夾爪現在位置
      OUT     M3002  ; 中心機光纖定位OK-2
337   LD      SM400
      +       D201 K5 D210
341   LD<     D3248 D3259  ; 拍板現在位置換算板寬
      OUT     M3005  ; 拍板馬達手動至內移定點_單邊ON
345   LD      X8D  ; 中心機左內光纖
      AND     X8E  ; 中心機右內光纖
      OR      M3006
      OUT     M3001  ; 中心機拍板減速光纖定位OK
349   LD      M3000  ; 中心機光纖定位OK-1
      MEP
      ANI     Y0A2A  ; #2 AXIS JOG+
      ANI     Y0A2B  ; #2 AXIS JOG-
      DMOV    D3248 D3270  ; 拍板現在位置換算板寬暫存
355   LD      SM400
      D/      D3248 K10 D3272  ; 拍板現在位置換算板寬暫存
360   LDP     M2607  ; 拍板一行程PB
      OR      T613
      ANI     M2613  ; 拍板馬達手動至內移定點KP
      ANI     M2619  ; 拍板一行程_拍板完成KP
      AND     M2000  ; 軸1伺服馬達外極限
      ANI     Y305  ; 進料ROBOT至取板下降位置-IN6
      OUT     M2617  ; 拍板一行程KP
368   LD      M3000  ; 中心機光纖定位OK-1
      OR      M2618  ; 拍板一行程_拍板OK
      AND     M2613  ; 拍板馬達手動至內移定點KP
      OUT     M2618  ; 拍板一行程_拍板OK
      AND     X3B  ; 中心機前夾爪-夾定點
      OUT     T57 K3
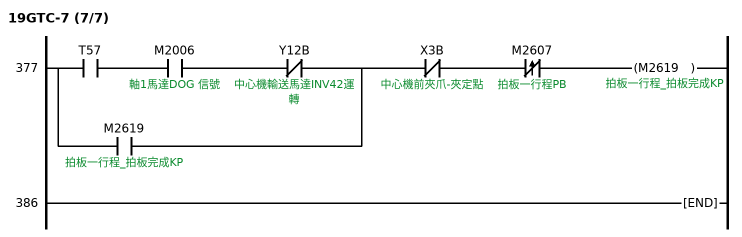
377   LD      T57
      AND     M2006  ; 軸1馬達DOG 信號
      ANI     Y12B  ; 中心機輸送馬達INV42運轉
      OR      M2619  ; 拍板一行程_拍板完成KP
      ANI     X3B  ; 中心機前夾爪-夾定點
      ANDPI   M2607  ; 拍板一行程PB
      OUT     M2619  ; 拍板一行程_拍板完成KP
386   END
END_PROGRAM

PROGRAM 20TEST
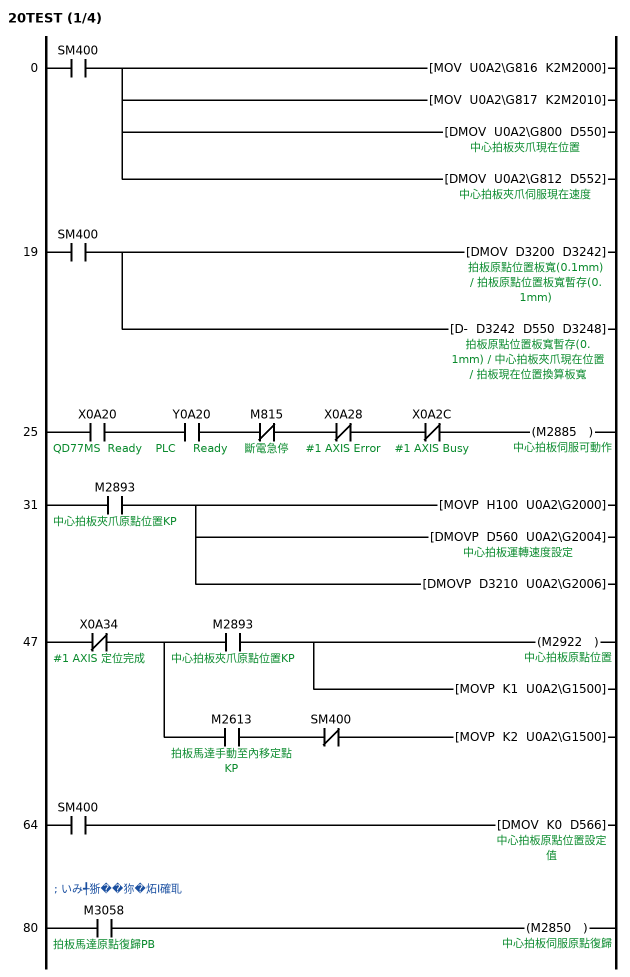
0     LD      SM400
      MOV     U0A2\G816 K2M2000  ; 軸1伺服馬達外極限
      MOV     U0A2\G817 K2M2010  ; Axis01  速度控制
      DMOV    U0A2\G800 D550  ; 中心拍板夾爪現在位置
      DMOV    U0A2\G812 D552  ; 中心拍板夾爪伺服現在速度
19    LD      SM400
      DMOV    D3200 D3242  ; 拍板原點位置板寬(0.1mm) / 拍板原點位置板寬暫存(0.1mm)
      D-      D3242 D550 D3248  ; 拍板現在位置換算板寬
25    LD      X0A20  ; QD77MS  Ready
      AND     Y0A20  ; PLC     Ready
      ANI     M815  ; 斷電急停
      ANI     X0A28  ; #1 AXIS Error
      ANI     X0A2C  ; #1 AXIS Busy
      OUT     M2885  ; 中心拍板伺服可動作
31    LD      M2893  ; 中心拍板夾爪原點位置KP
      MOVP    H100 U0A2\G2000
      DMOVP   D560 U0A2\G2004  ; 中心拍板運轉速度設定
      DMOVP   D3210 U0A2\G2006
47    LDI     X0A34  ; #1 AXIS 定位完成
      MPS
      AND     M2893  ; 中心拍板夾爪原點位置KP
      OUT     M2922  ; 中心拍板原點位置
      MOVP    K1 U0A2\G1500
      MPP
      AND     M2613  ; 拍板馬達手動至內移定點KP
      ANI     SM400
      MOVP    K2 U0A2\G1500
64    LD      SM400
      DMOV    K0 D566  ; 中心拍板原點位置設定值
; 中心拍板伺服原點復歸
80    LD      M3058  ; 拍板馬達原點復歸PB
      OUT     M2850  ; 中心拍板伺服原點復歸
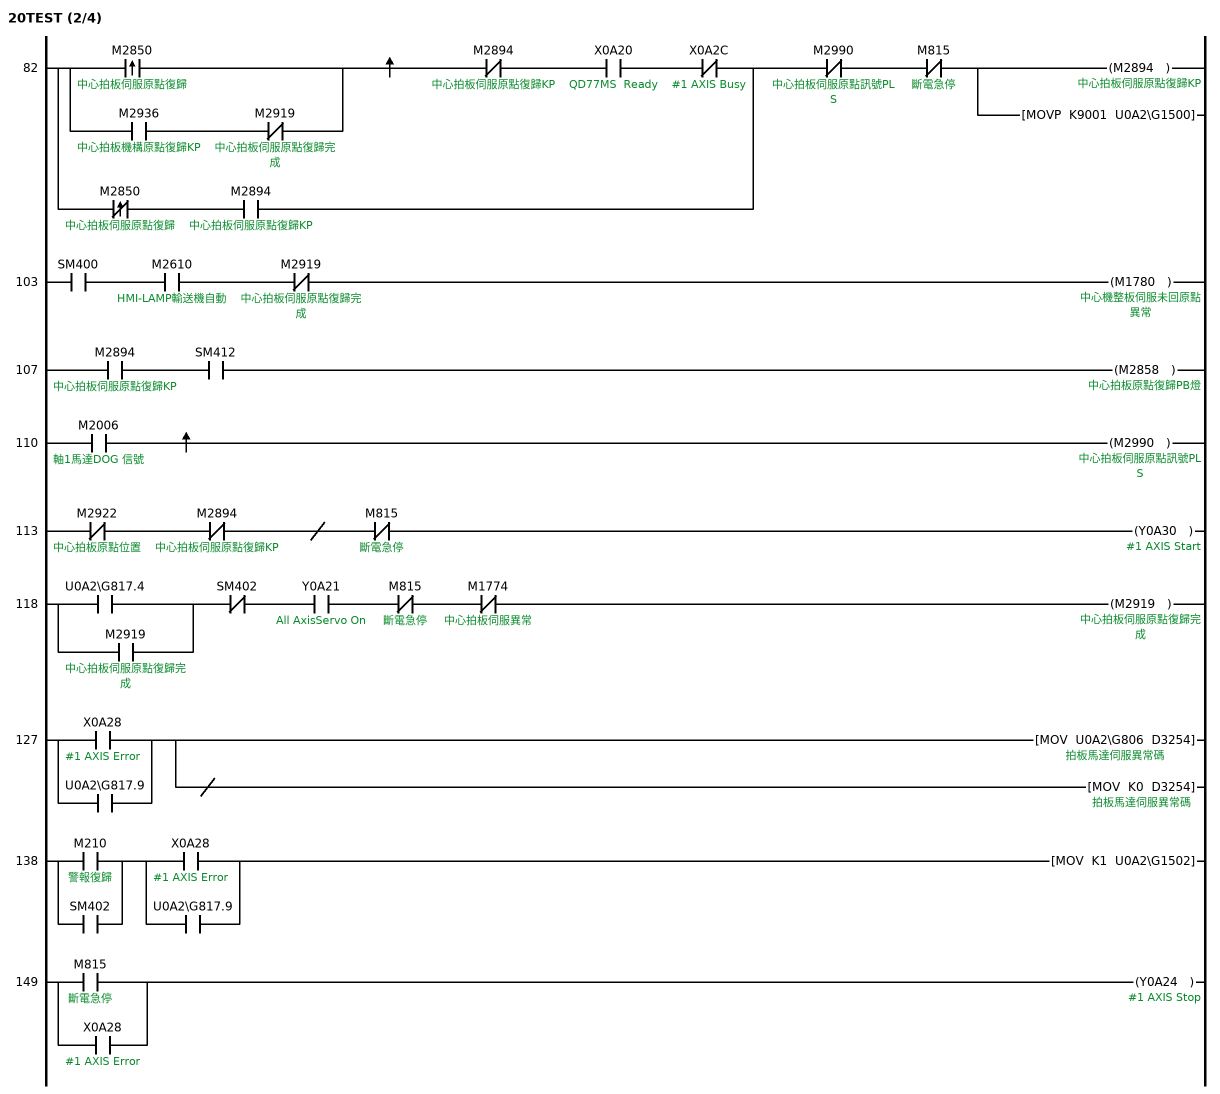
82    LDP     M2850  ; 中心拍板伺服原點復歸
      LD      M2936  ; 中心拍板機構原點復歸KP
      ANI     M2919  ; 中心拍板伺服原點復歸完成
      ORB
      MEP
      ANI     M2894  ; 中心拍板伺服原點復歸KP
      AND     X0A20  ; QD77MS  Ready
      ANI     X0A2C  ; #1 AXIS Busy
      LDPI    M2850  ; 中心拍板伺服原點復歸
      AND     M2894  ; 中心拍板伺服原點復歸KP
      ORB
      ANI     M2990  ; 中心拍板伺服原點訊號PLS
      ANI     M815  ; 斷電急停
      OUT     M2894  ; 中心拍板伺服原點復歸KP
      MOVP    K9001 U0A2\G1500
103   LD      SM400
      AND     M2610  ; HMI-LAMP輸送機自動
      ANI     M2919  ; 中心拍板伺服原點復歸完成
      OUT     M1780  ; 中心機整板伺服未回原點異常
107   LD      M2894  ; 中心拍板伺服原點復歸KP
      AND     SM412
      OUT     M2858  ; 中心拍板原點復歸PB燈
110   LD      M2006  ; 軸1馬達DOG 信號
      MEP
      OUT     M2990  ; 中心拍板伺服原點訊號PLS
113   LDI     M2922  ; 中心拍板原點位置
      ANI     M2894  ; 中心拍板伺服原點復歸KP
      INV
      ANI     M815  ; 斷電急停
      OUT     Y0A30  ; #1 AXIS Start
118   LD      U0A2\G817.4
      OR      M2919  ; 中心拍板伺服原點復歸完成
      ANI     SM402
      AND     Y0A21  ; All AxisServo On
      ANI     M815  ; 斷電急停
      ANI     M1774  ; 中心拍板伺服異常
      OUT     M2919  ; 中心拍板伺服原點復歸完成
127   LD      X0A28  ; #1 AXIS Error
      OR      U0A2\G817.9
      MOV     U0A2\G806 D3254  ; 拍板馬達伺服異常碼
      INV
      MOV     K0 D3254
138   LD      M210  ; 警報復歸
      OR      SM402
      LD      X0A28  ; #1 AXIS Error
      OR      U0A2\G817.9
      ANB
      MOV     K1 U0A2\G1502
149   LD      M815  ; 斷電急停
      OR      X0A28  ; #1 AXIS Error
      OUT     Y0A24  ; #1 AXIS Stop
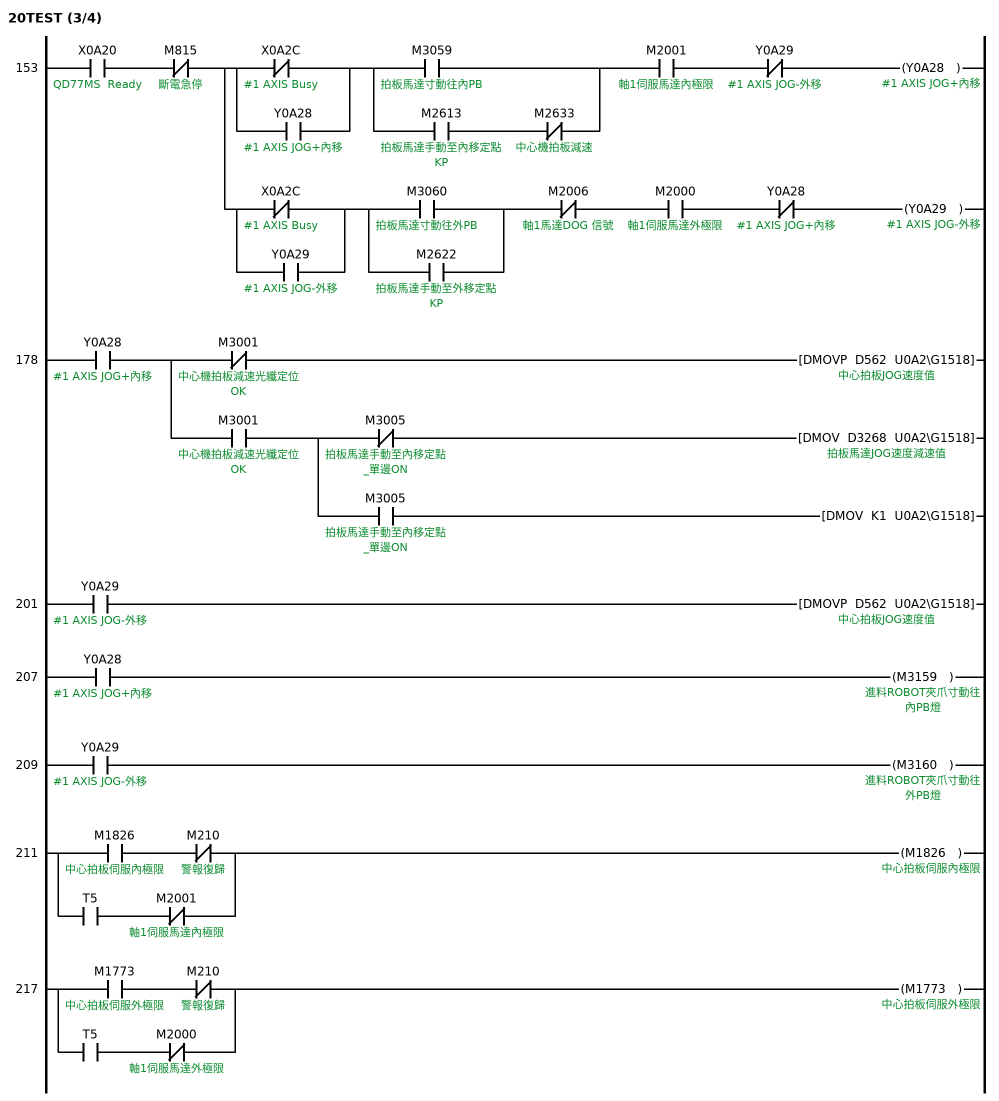
153   LD      X0A20  ; QD77MS  Ready
      ANI     M815  ; 斷電急停
      MPS
      LDI     X0A2C  ; #1 AXIS Busy
      OR      Y0A28  ; #1 AXIS JOG+內移
      ANB
      LD      M3059  ; 拍板馬達寸動往內PB
      LD      M2613  ; 拍板馬達手動至內移定點KP
      ANI     M2633  ; 中心機拍板減速
      ORB
      ANB
      AND     M2001  ; 軸1伺服馬達內極限
      ANI     Y0A29  ; #1 AXIS JOG-外移
      OUT     Y0A28  ; #1 AXIS JOG+內移
      MPP
      LDI     X0A2C  ; #1 AXIS Busy
      OR      Y0A29  ; #1 AXIS JOG-外移
      ANB
      LD      M3060  ; 拍板馬達寸動往外PB
      OR      M2622  ; 拍板馬達手動至外移定點KP
      ANB
      ANI     M2006  ; 軸1馬達DOG 信號
      AND     M2000  ; 軸1伺服馬達外極限
      ANI     Y0A28  ; #1 AXIS JOG+內移
      OUT     Y0A29  ; #1 AXIS JOG-外移
178   LD      Y0A28  ; #1 AXIS JOG+內移
      MPS
      ANI     M3001  ; 中心機拍板減速光纖定位OK
      DMOVP   D562 U0A2\G1518  ; 中心拍板JOG速度值
      MPP
      AND     M3001  ; 中心機拍板減速光纖定位OK
      MPS
      ANI     M3005  ; 拍板馬達手動至內移定點_單邊ON
      DMOV    D3268 U0A2\G1518  ; 拍板馬達JOG速度減速值
      MPP
      AND     M3005  ; 拍板馬達手動至內移定點_單邊ON
      DMOV    K1 U0A2\G1518
201   LD      Y0A29  ; #1 AXIS JOG-外移
      DMOVP   D562 U0A2\G1518
207   LD      Y0A28  ; #1 AXIS JOG+內移
      OUT     M3159  ; 進料ROBOT夾爪寸動往內PB燈
209   LD      Y0A29  ; #1 AXIS JOG-外移
      OUT     M3160  ; 進料ROBOT夾爪寸動往外PB燈
211   LD      M1826  ; 中心拍板伺服內極限
      ANI     M210  ; 警報復歸
      LD      T5
      ANI     M2001  ; 軸1伺服馬達內極限
      ORB
      OUT     M1826  ; 中心拍板伺服內極限
217   LD      M1773  ; 中心拍板伺服外極限
      ANI     M210  ; 警報復歸
      LD      T5
      ANI     M2000  ; 軸1伺服馬達外極限
      ORB
      OUT     M1773  ; 中心拍板伺服外極限
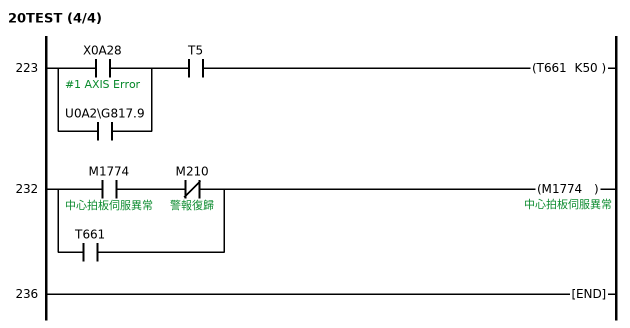
223   LD      X0A28  ; #1 AXIS Error
      OR      U0A2\G817.9
      AND     T5
      OUT     T661 K50
232   LD      M1774  ; 中心拍板伺服異常
      ANI     M210  ; 警報復歸
      OR      T661
      OUT     M1774  ; 中心拍板伺服異常
236   END
END_PROGRAM

PROGRAM 22PB
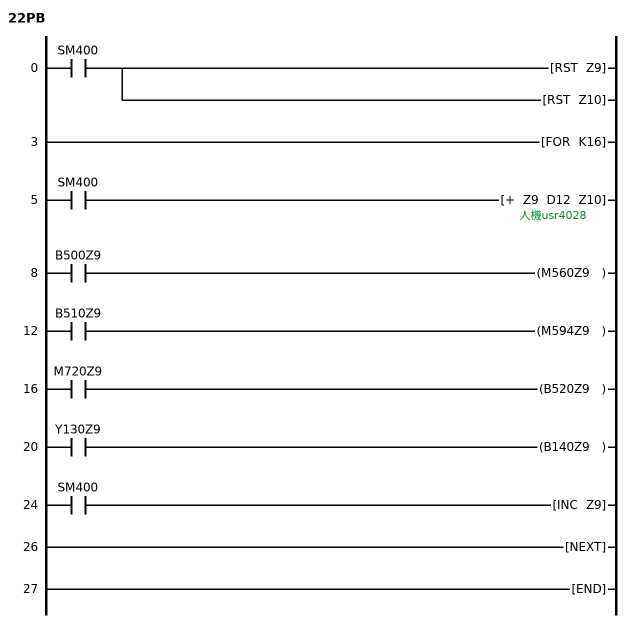
0     LD      SM400
      RST     Z9
      RST     Z10
3     FOR     K16
5     LD      SM400
      +       Z9 D12 Z10  ; 人機usr4028
8     LD      B500Z9
      OUT     M560Z9
12    LD      B510Z9
      OUT     M594Z9
16    LD      M720Z9
      OUT     B520Z9
20    LD      Y130Z9
      OUT     B140Z9
24    LD      SM400
      INC     Z9
26    NEXT
27    END
END_PROGRAM

PROGRAM MAIN
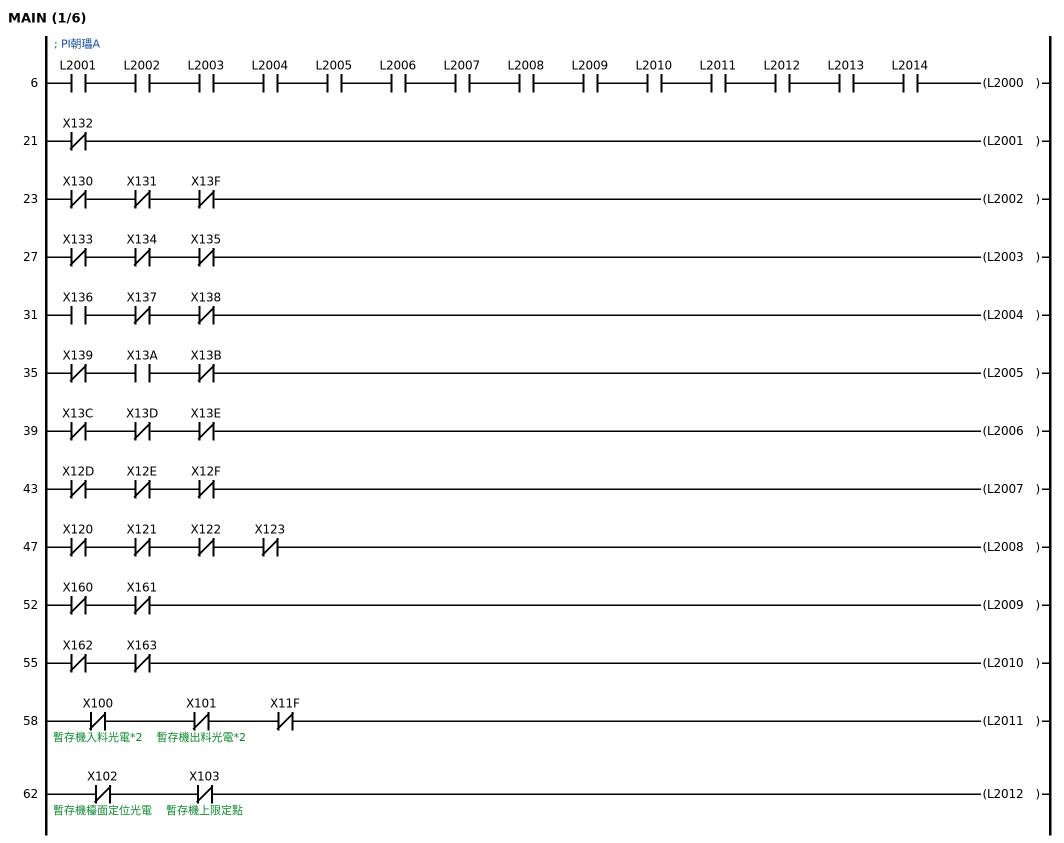
; PI朝瓃Α
6     LD      L2001
      AND     L2002
      AND     L2003
      AND     L2004
      AND     L2005
      AND     L2006
      AND     L2007
      AND     L2008
      AND     L2009
      AND     L2010
      AND     L2011
      AND     L2012
      AND     L2013
      AND     L2014
      OUT     L2000
21    LDI     X132
      OUT     L2001
23    LDI     X130
      ANI     X131
      ANI     X13F
      OUT     L2002
27    LDI     X133
      ANI     X134
      ANI     X135
      OUT     L2003
31    LD      X136
      ANI     X137
      ANI     X138
      OUT     L2004
35    LDI     X139
      AND     X13A
      ANI     X13B
      OUT     L2005
39    LDI     X13C
      ANI     X13D
      ANI     X13E
      OUT     L2006
43    LDI     X12D
      ANI     X12E
      ANI     X12F
      OUT     L2007
47    LDI     X120
      ANI     X121
      ANI     X122
      ANI     X123
      OUT     L2008
52    LDI     X160
      ANI     X161
      OUT     L2009
55    LDI     X162
      ANI     X163
      OUT     L2010
58    LDI     X100  ; 暫存機入料光電*2
      ANI     X101  ; 暫存機出料光電*2
      ANI     X11F
      OUT     L2011
62    LDI     X102  ; 暫存機檯面定位光電
      ANI     X103  ; 暫存機上限定點
      OUT     L2012
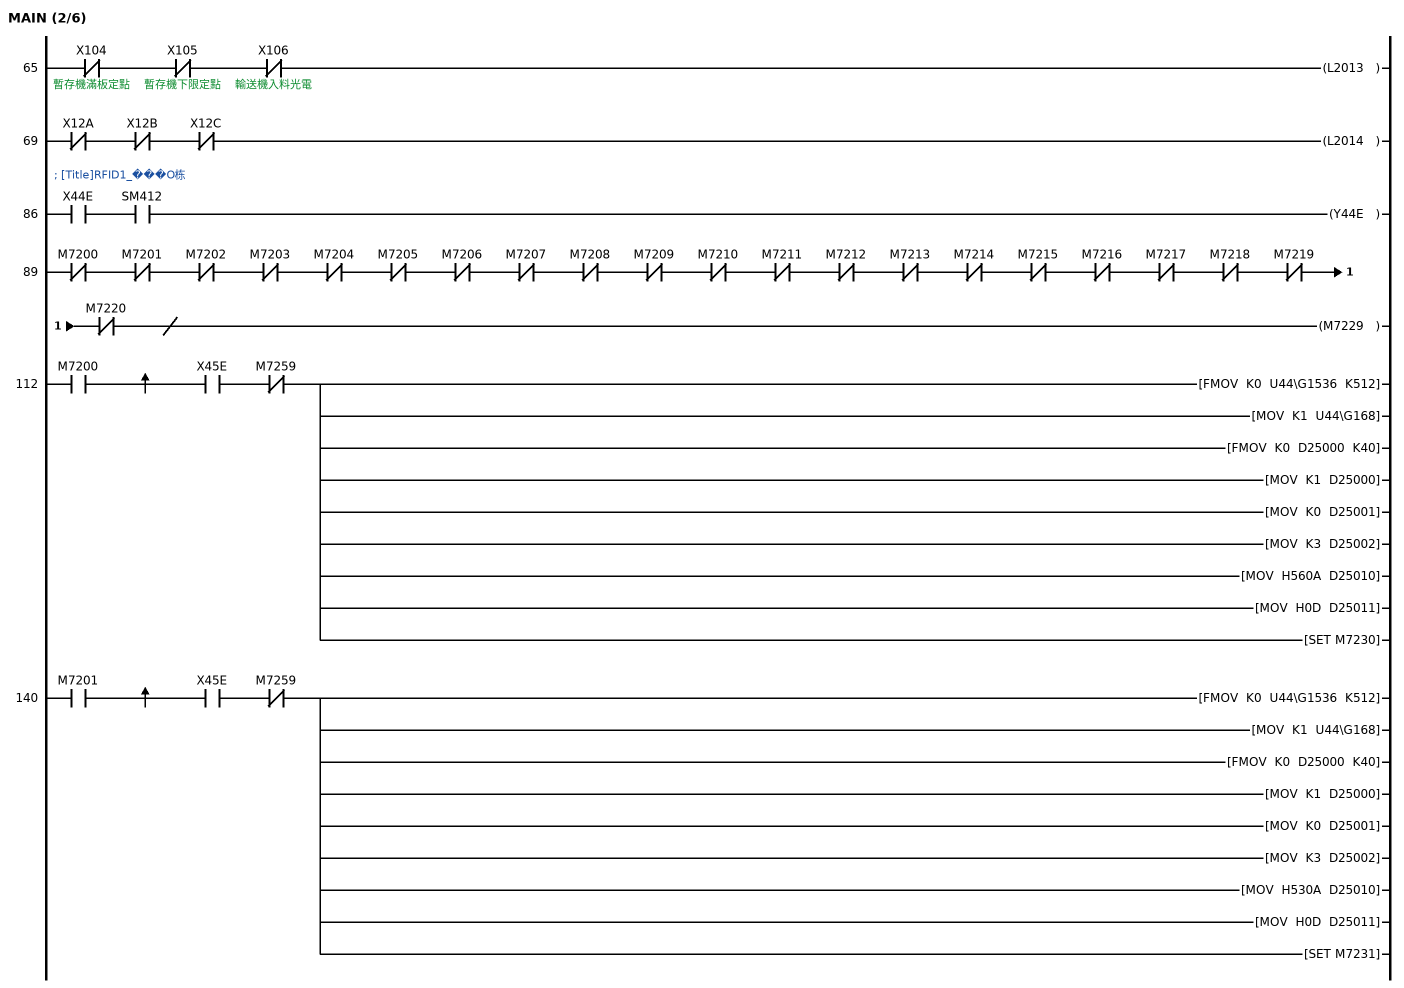
65    LDI     X104  ; 暫存機滿板定點
      ANI     X105  ; 暫存機下限定點
      ANI     X106  ; 輸送機入料光電
      OUT     L2013
69    LDI     X12A
      ANI     X12B
      ANI     X12C
      OUT     L2014
; [Title]RFID1_指令集
86    LD      X44E
      AND     SM412
      OUT     Y44E
89    LDI     M7200
      ANI     M7201
      ANI     M7202
      ANI     M7203
      ANI     M7204
      ANI     M7205
      ANI     M7206
      ANI     M7207
      ANI     M7208
      ANI     M7209
      ANI     M7210
      ANI     M7211
      ANI     M7212
      ANI     M7213
      ANI     M7214
      ANI     M7215
      ANI     M7216
      ANI     M7217
      ANI     M7218
      ANI     M7219
      ANI     M7220
      INV
      OUT     M7229
112   LD      M7200
      MEP
      AND     X45E
      ANI     M7259
      FMOV    K0 U44\G1536 K512
      MOV     K1 U44\G168
      FMOV    K0 D25000 K40
      MOV     K1 D25000
      MOV     K0 D25001
      MOV     K3 D25002
      MOV     H560A D25010
      MOV     H0D D25011
      SET     M7230
140   LD      M7201
      MEP
      AND     X45E
      ANI     M7259
      FMOV    K0 U44\G1536 K512
      MOV     K1 U44\G168
      FMOV    K0 D25000 K40
      MOV     K1 D25000
      MOV     K0 D25001
      MOV     K3 D25002
      MOV     H530A D25010
      MOV     H0D D25011
      SET     M7231
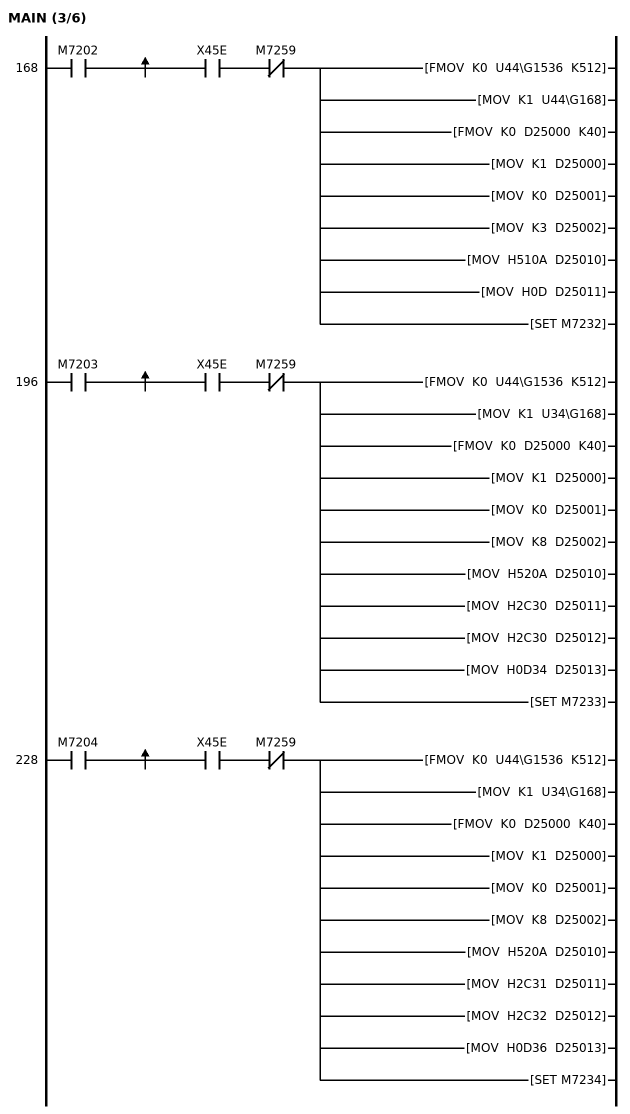
168   LD      M7202
      MEP
      AND     X45E
      ANI     M7259
      FMOV    K0 U44\G1536 K512
      MOV     K1 U44\G168
      FMOV    K0 D25000 K40
      MOV     K1 D25000
      MOV     K0 D25001
      MOV     K3 D25002
      MOV     H510A D25010
      MOV     H0D D25011
      SET     M7232
196   LD      M7203
      MEP
      AND     X45E
      ANI     M7259
      FMOV    K0 U44\G1536 K512
      MOV     K1 U34\G168
      FMOV    K0 D25000 K40
      MOV     K1 D25000
      MOV     K0 D25001
      MOV     K8 D25002
      MOV     H520A D25010
      MOV     H2C30 D25011
      MOV     H2C30 D25012
      MOV     H0D34 D25013
      SET     M7233
228   LD      M7204
      MEP
      AND     X45E
      ANI     M7259
      FMOV    K0 U44\G1536 K512
      MOV     K1 U34\G168
      FMOV    K0 D25000 K40
      MOV     K1 D25000
      MOV     K0 D25001
      MOV     K8 D25002
      MOV     H520A D25010
      MOV     H2C31 D25011
      MOV     H2C32 D25012
      MOV     H0D36 D25013
      SET     M7234
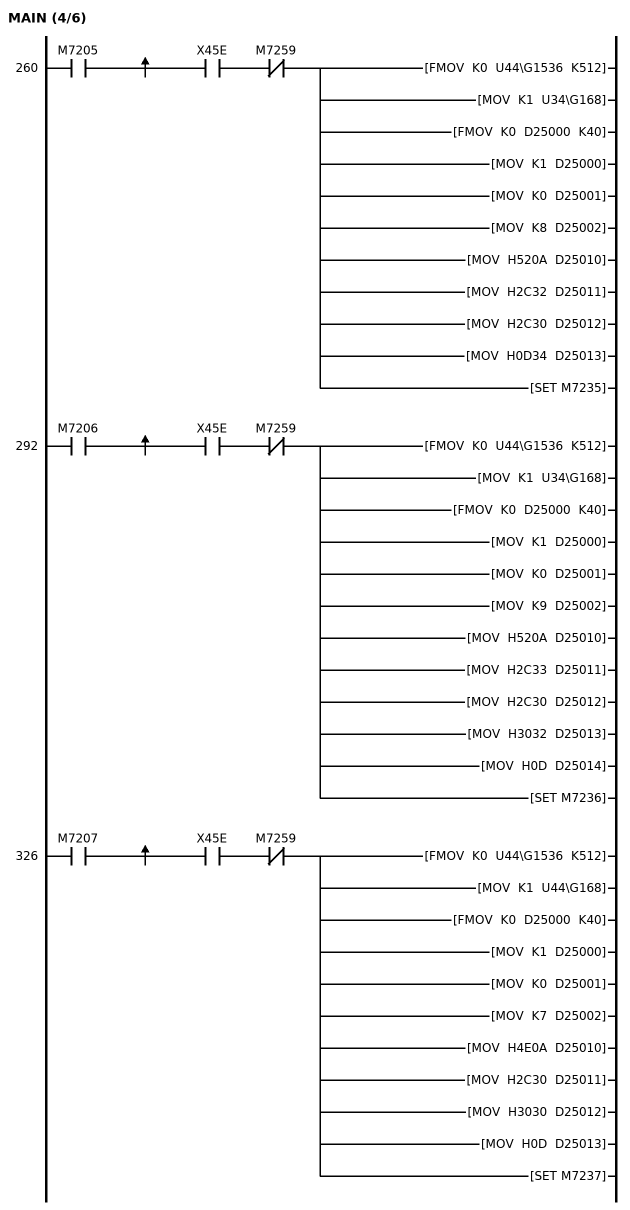
260   LD      M7205
      MEP
      AND     X45E
      ANI     M7259
      FMOV    K0 U44\G1536 K512
      MOV     K1 U34\G168
      FMOV    K0 D25000 K40
      MOV     K1 D25000
      MOV     K0 D25001
      MOV     K8 D25002
      MOV     H520A D25010
      MOV     H2C32 D25011
      MOV     H2C30 D25012
      MOV     H0D34 D25013
      SET     M7235
292   LD      M7206
      MEP
      AND     X45E
      ANI     M7259
      FMOV    K0 U44\G1536 K512
      MOV     K1 U34\G168
      FMOV    K0 D25000 K40
      MOV     K1 D25000
      MOV     K0 D25001
      MOV     K9 D25002
      MOV     H520A D25010
      MOV     H2C33 D25011
      MOV     H2C30 D25012
      MOV     H3032 D25013
      MOV     H0D D25014
      SET     M7236
326   LD      M7207
      MEP
      AND     X45E
      ANI     M7259
      FMOV    K0 U44\G1536 K512
      MOV     K1 U44\G168
      FMOV    K0 D25000 K40
      MOV     K1 D25000
      MOV     K0 D25001
      MOV     K7 D25002
      MOV     H4E0A D25010
      MOV     H2C30 D25011
      MOV     H3030 D25012
      MOV     H0D D25013
      SET     M7237
